  MoveL 9104 to (-26.02, -28.9, -15.5) mm, rotated rx -180 ry 0 rz 90 deg; joints [72.625, -17.388, 85.354, 0, 22.034, 72.625]
  MoveL 9105 to (-25.99, -28.43, -15.5) mm, rotated rx 180 ry 0 rz 90 deg; joints [72.641, -17.39, 85.362, 0, 22.028, 72.641]
  MoveC 9106 to (-26.88, -26.52, -15.5) mm, rotated rx -180 ry 0 rz 90 deg; joints [72.694, -17.416, 85.465, 0, 21.951, 72.694] to (-28.69, -25.44, -15.5) mm, rotated rx 180 ry 0 rz 90 deg; joints [72.71, -17.453, 85.614, 0, 21.839, 72.71]
  MoveL 9107 to (-30.8, -25.8, -15.5) mm, rotated rx 180 ry 0 rz 90 deg; joints [72.677, -17.487, 85.752, 0, 21.735, 72.677]
  MoveL 9108 to (-42.04, -27.96, -15.5) mm, rotated rx 180 ry 0 rz 90 deg; joints [72.492, -17.665, 86.481, 0, 21.184, 72.492]
  MoveL 9109 to (-45.96, -28.7, -15.5) mm, rotated rx -180 ry 0 rz 90 deg; joints [72.427, -17.726, 86.733, 0, 20.993, 72.427]
  MoveL 9110 to (-48.22, -29.15, -15.5) mm, rotated rx -180 ry 0 rz 90 deg; joints [72.389, -17.761, 86.878, 0, 20.882, 72.389]
  MoveL 9111 to (-46.77, -36.56, -15.5) mm, rotated rx -180 ry 0 rz 90 deg; joints [72.161, -17.698, 86.617, 0, 21.081, 72.161]
  MoveL 9112 to (-46.77, -36.56, -12.5) mm, rotated rx -180 ry 0 rz 90 deg; joints [72.161, -17.853, 86.72, 0, 21.133, 72.161]
  Establecer velocidad (1000.0 mm/s)
  MoveL 9113 to (-46.77, -36.56, 10) mm, rotated rx 180 ry 0 rz 90 deg; joints [72.161, -19.016, 87.475, 0, 21.541, 72.161]
  Establecer velocidad (66.7 mm/s)
  MoveL 9114 to (-40.09, -36.12, 10) mm, rotated rx -180 ry 0 rz 90 deg; joints [72.245, -18.904, 87.027, 0, 21.878, 72.245]
  MoveL 9115 to (-40.09, -36.12, -12.5) mm, rotated rx -180 ry 0 rz 90 deg; joints [72.245, -17.744, 86.271, 0, 21.473, 72.245]
  MoveL 9116 to (-40.2, -34.6, -12.91) mm, rotated rx 180 ry 0 rz 90 deg; joints [72.294, -17.733, 86.298, 0, 21.435, 72.294]
  MoveL 9117 to (-40.67, -33.16, -13.31) mm, rotated rx 180 ry 0 rz 90 deg; joints [72.336, -17.728, 86.348, 0, 21.379, 72.336]
  MoveL 9118 to (-41.45, -31.85, -13.72) mm, rotated rx -180 ry 0 rz 90 deg; joints [72.371, -17.727, 86.416, 0, 21.31, 72.371]
  MoveL 9119 to (-42.49, -30.75, -14.12) mm, rotated rx -180 ry 0 rz 90 deg; joints [72.396, -17.729, 86.498, 0, 21.231, 72.396]
  MoveL 9120 to (-43.76, -29.91, -14.53) mm, rotated rx -180 ry 0 rz 90 deg; joints [72.41, -17.733, 86.589, 0, 21.144, 72.41]
  MoveL 9121 to (-45.18, -29.37, -14.94) mm, rotated rx 180 ry 0 rz 90 deg; joints [72.413, -17.739, 86.685, 0, 21.054, 72.413]
  MoveL 9122 to (-46.68, -29.16, -15.34) mm, rotated rx 180 ry 0 rz 90 deg; joints [72.404, -17.743, 86.778, 0, 20.965, 72.404]
  MoveL 9123 to (-48.19, -29.31, -15.75) mm, rotated rx 180 ry 0 rz 90 deg; joints [72.384, -17.746, 86.864, 0, 20.882, 72.384]
  MoveC 9124 to (-48.97, -29.46, -15.75) mm, rotated rx -180 ry 0 rz 90 deg; joints [72.37, -17.758, 86.914, 0, 20.844, 72.37] to (-49.75, -29.62, -15.75) mm, rotated rx 180 ry 0 rz 90 deg; joints [72.357, -17.77, 86.964, 0, 20.807, 72.357]
  MoveL 9125 to (-52.59, -30.15, -15.75) mm, rotated rx -180 ry 0 rz 90 deg; joints [72.31, -17.813, 87.146, 0, 20.668, 72.31]
  MoveL 9126 to (-67.59, -33.11, -15.75) mm, rotated rx 180 ry 0 rz 90 deg; joints [72.054, -18.036, 88.096, 0, 19.939, 72.054]
  MoveC 9127 to (-68.93, -33.88, -15.75) mm, rotated rx -180 ry 0 rz 90 deg; joints [72.014, -18.053, 88.169, 0, 19.883, 72.014] to (-69.53, -35.3, -15.75) mm, rotated rx 180 ry 0 rz 90 deg; joints [71.96, -18.055, 88.179, 0, 19.876, 71.96]
  MoveC 9128 to (-69.55, -35.58, -15.75) mm, rotated rx -180 ry 0 rz 90 deg; joints [71.951, -18.053, 88.174, 0, 19.88, 71.951] to (-69.55, -35.85, -15.75) mm, rotated rx 180 ry 0 rz 90 deg; joints [71.942, -18.052, 88.168, 0, 19.884, 71.942]
  MoveL 9129 to (-69.55, -65.86, -15.75) mm, rotated rx 180 ry 0 rz 90 deg; joints [70.954, -17.895, 87.491, 0, 20.404, 70.954]
  MoveL 9130 to (-69.55, -66.98, -15.75) mm, rotated rx 180 ry 0 rz 90 deg; joints [70.918, -17.889, 87.465, 0, 20.424, 70.918]
  MoveC 9131 to (-68.8, -68.74, -15.75) mm, rotated rx 180 ry 0 rz 90 deg; joints [70.869, -17.867, 87.373, 0, 20.494, 70.869] to (-67.01, -69.45, -15.75) mm, rotated rx 180 ry 0 rz 90 deg; joints [70.866, -17.835, 87.236, 0, 20.599, 70.866]
  MoveC 9132 to (-52.7, -69.11, -15.75) mm, rotated rx -180 ry 0 rz 90 deg; joints [71.037, -17.604, 86.273, 0, 21.33, 71.037] to (-38.38, -68.71, -15.75) mm, rotated rx -180 ry 0 rz 90 deg; joints [71.208, -17.364, 85.301, 0, 22.063, 71.208]
  MoveC 9133 to (-36.78, -68.19, -15.75) mm, rotated rx 180 ry 0 rz 90 deg; joints [71.242, -17.339, 85.203, 0, 22.137, 71.242] to (-35.83, -66.81, -15.75) mm, rotated rx 180 ry 0 rz 90 deg; joints [71.297, -17.331, 85.169, 0, 22.162, 71.297]
  MoveL 9134 to (-26.19, -28.9, -15.75) mm, rotated rx 180 ry 0 rz 90 deg; joints [72.623, -17.378, 85.357, 0, 22.021, 72.623]
  MoveC 9135 to (-26.99, -26.82, -15.75) mm, rotated rx 180 ry 0 rz 90 deg; joints [72.683, -17.403, 85.458, 0, 21.945, 72.683] to (-28.9, -25.65, -15.75) mm, rotated rx 180 ry 0 rz 90 deg; joints [72.701, -17.442, 85.616, 0, 21.827, 72.701]
  MoveC 9136 to (-38.55, -27.45, -15.75) mm, rotated rx -180 ry 0 rz 90 deg; joints [72.544, -17.597, 86.243, 0, 21.353, 72.544] to (-48.19, -29.31, -15.75) mm, rotated rx 180 ry 0 rz 90 deg; joints [72.384, -17.746, 86.864, 0, 20.882, 72.384]
  MoveL 9137 to (-46.74, -36.72, -15.75) mm, rotated rx 180 ry 0 rz 90 deg; joints [72.156, -17.684, 86.603, 0, 21.081, 72.156]
  MoveL 9138 to (-46.74, -36.72, -12.75) mm, rotated rx -180 ry 0 rz 90 deg; joints [72.156, -17.839, 86.705, 0, 21.133, 72.156]
  Establecer velocidad (1000.0 mm/s)
  MoveL 9139 to (-46.74, -36.72, 10) mm, rotated rx 180 ry 0 rz 90 deg; joints [72.156, -19.014, 87.469, 0, 21.545, 72.156]
  Establecer velocidad (66.7 mm/s)
  MoveL 9140 to (-61.31, 35.31, 10) mm, rotated rx -180 ry 0 rz 90 deg; joints [74.405, -19.6, 89.929, 0, 19.671, 74.405]
  MoveL 9141 to (-61.31, 35.31, -12.5) mm, rotated rx -180 ry 0 rz 90 deg; joints [74.405, -18.425, 89.173, 0, 19.251, 74.405]
  MoveL 9142 to (-62.81, 35.49, -12.91) mm, rotated rx 180 ry 0 rz 90 deg; joints [74.397, -18.427, 89.265, 0, 19.162, 74.397]
  MoveL 9143 to (-64.32, 35.31, -13.31) mm, rotated rx 180 ry 0 rz 90 deg; joints [74.377, -18.427, 89.349, 0, 19.079, 74.377]
  MoveL 9144 to (-65.75, 34.8, -13.72) mm, rotated rx -180 ry 0 rz 90 deg; joints [74.346, -18.425, 89.421, 0, 19.004, 74.346]
  MoveL 9145 to (-67.04, 33.98, -14.12) mm, rotated rx -180 ry 0 rz 90 deg; joints [74.306, -18.42, 89.478, 0, 18.941, 74.306]
  MoveL 9146 to (-68.11, 32.9, -14.53) mm, rotated rx 180 ry 0 rz 90 deg; joints [74.259, -18.41, 89.516, 0, 18.894, 74.259]
  MoveL 9147 to (-68.91, 31.61, -14.94) mm, rotated rx -180 ry 0 rz 90 deg; joints [74.208, -18.395, 89.531, 0, 18.864, 74.208]
  MoveL 9148 to (-69.41, 30.18, -15.34) mm, rotated rx 180 ry 0 rz 90 deg; joints [74.154, -18.375, 89.524, 0, 18.851, 74.154]
  MoveL 9149 to (-69.55, 28.67, -15.75) mm, rotated rx 180 ry 0 rz 90 deg; joints [74.102, -18.349, 89.49, 0, 18.859, 74.102]
  MoveL 9150 to (-69.55, 5.69, -15.75) mm, rotated rx -180 ry 0 rz 90 deg; joints [73.327, -18.25, 89.04, 0, 19.21, 73.327]
  MoveC 9151 to (-68.75, 3.78, -15.75) mm, rotated rx 180 ry 0 rz 90 deg; joints [73.271, -18.229, 88.948, 0, 19.281, 73.271] to (-66.81, 3.09, -15.75) mm, rotated rx 180 ry 0 rz 90 deg; joints [73.267, -18.197, 88.804, 0, 19.393, 73.267]
  MoveL 9152 to (-65.86, 3.29, -15.75) mm, rotated rx 180 ry 0 rz 90 deg; joints [73.283, -18.183, 88.744, 0, 19.439, 73.283]
  MoveL 9153 to (-62.19, 4.19, -15.75) mm, rotated rx -180 ry 0 rz 90 deg; joints [73.35, -18.131, 88.515, 0, 19.616, 73.35]
  MoveC 9154 to (-44.56, 8.55, -15.75) mm, rotated rx 180 ry 0 rz 90 deg; joints [73.67, -17.875, 87.406, 0, 20.469, 73.67] to (-26.96, 13.02, -15.75) mm, rotated rx 180 ry 0 rz 90 deg; joints [73.986, -17.606, 86.283, 0, 21.323, 73.986]
  MoveC 9155 to (-26.48, 13.21, -15.75) mm, rotated rx -180 ry 0 rz 90 deg; joints [73.997, -17.599, 86.254, 0, 21.345, 73.997] to (-26.06, 13.5, -15.75) mm, rotated rx 180 ry 0 rz 90 deg; joints [74.01, -17.593, 86.231, 0, 21.363, 74.01]
  MoveC 9156 to (-25.23, 14.68, -15.75) mm, rotated rx -180 ry 0 rz 90 deg; joints [74.057, -17.585, 86.197, 0, 21.389, 74.057] to (-25.03, 16.11, -15.75) mm, rotated rx 180 ry 0 rz 90 deg; joints [74.106, -17.589, 86.211, 0, 21.378, 74.106]
  MoveC 9157 to (-25.09, 16.38, -15.75) mm, rotated rx 180 ry 0 rz 90 deg; joints [74.114, -17.591, 86.22, 0, 21.371, 74.114] to (-25.17, 16.64, -15.75) mm, rotated rx 180 ry 0 rz 90 deg; joints [74.122, -17.594, 86.231, 0, 21.362, 74.122]
  MoveL 9158 to (-29.47, 28.93, -15.75) mm, rotated rx -180 ry 0 rz 90 deg; joints [74.488, -17.723, 86.768, 0, 20.955, 74.488]
  MoveC 9159 to (-29.9, 29.71, -15.75) mm, rotated rx 180 ry 0 rz 90 deg; joints [74.51, -17.734, 86.812, 0, 20.922, 74.51] to (-30.55, 30.32, -15.75) mm, rotated rx 180 ry 0 rz 90 deg; joints [74.525, -17.747, 86.869, 0, 20.879, 74.525]
  MoveC 9160 to (-48.17, 42.1, -15.75) mm, rotated rx 180 ry 0 rz 90 deg; joints [74.756, -18.082, 88.299, 0, 19.783, 74.756] to (-65.86, 53.77, -15.75) mm, rotated rx 180 ry 0 rz 90 deg; joints [74.989, -18.397, 89.708, 0, 18.689, 74.989]
  MoveC 9161 to (-67.73, 53.7, -15.75) mm, rotated rx 180 ry 0 rz 90 deg; joints [74.97, -18.424, 89.832, 0, 18.592, 74.97] to (-69.23, 52.59, -15.75) mm, rotated rx 180 ry 0 rz 90 deg; joints [74.918, -18.442, 89.913, 0, 18.529, 74.918]
  MoveC 9162 to (-69.47, 52.15, -15.75) mm, rotated rx 180 ry 0 rz 90 deg; joints [74.901, -18.443, 89.921, 0, 18.522, 74.901] to (-69.55, 51.65, -15.75) mm, rotated rx 180 ry 0 rz 90 deg; joints [74.883, -18.442, 89.917, 0, 18.525, 74.883]
  MoveL 9163 to (-69.55, 28.67, -15.75) mm, rotated rx 180 ry 0 rz 90 deg; joints [74.102, -18.349, 89.49, 0, 18.859, 74.102]
  MoveL 9164 to (-62, 28.67, -15.75) mm, rotated rx -180 ry 0 rz 90 deg; joints [74.174, -18.237, 88.983, 0, 19.254, 74.174]
  MoveL 9165 to (-62, 28.67, -12.75) mm, rotated rx 180 ry 0 rz 90 deg; joints [74.174, -18.394, 89.086, 0, 19.308, 74.174]
  Establecer velocidad (1000.0 mm/s)
  MoveL 9166 to (-62, 28.67, 10) mm, rotated rx 180 ry 0 rz 90 deg; joints [74.174, -19.582, 89.85, 0, 19.732, 74.174]
  Establecer velocidad (66.7 mm/s)
  MoveL 9167 to (-61.15, 35.31, 10) mm, rotated rx 180 ry 0 rz 90 deg; joints [74.407, -19.598, 89.918, 0, 19.679, 74.407]
  MoveL 9168 to (-61.15, 35.31, -12.75) mm, rotated rx 180 ry 0 rz 90 deg; joints [74.407, -18.409, 89.154, 0, 19.255, 74.407]
  MoveL 9169 to (-62.65, 35.49, -13.16) mm, rotated rx -180 ry 0 rz 90 deg; joints [74.399, -18.411, 89.245, 0, 19.166, 74.399]
  MoveL 9170 to (-64.16, 35.31, -13.56) mm, rotated rx 180 ry 0 rz 90 deg; joints [74.378, -18.412, 89.329, 0, 19.083, 74.378]
  MoveL 9171 to (-65.59, 34.8, -13.97) mm, rotated rx -180 ry 0 rz 90 deg; joints [74.347, -18.41, 89.402, 0, 19.008, 74.347]
  MoveL 9172 to (-66.87, 33.98, -14.37) mm, rotated rx 180 ry 0 rz 90 deg; joints [74.308, -18.404, 89.459, 0, 18.945, 74.308]
  MoveL 9173 to (-67.94, 32.9, -14.78) mm, rotated rx -180 ry 0 rz 90 deg; joints [74.261, -18.394, 89.496, 0, 18.898, 74.261]
  MoveL 9174 to (-68.75, 31.61, -15.19) mm, rotated rx -180 ry 0 rz 90 deg; joints [74.209, -18.379, 89.512, 0, 18.868, 74.209]
  MoveL 9175 to (-69.25, 30.18, -15.59) mm, rotated rx 180 ry 0 rz 90 deg; joints [74.156, -18.359, 89.504, 0, 18.856, 74.156]
  MoveL 9176 to (-69.39, 28.67, -16) mm, rotated rx -180 ry 0 rz 90 deg; joints [74.104, -18.334, 89.471, 0, 18.863, 74.104]
  MoveL 9177 to (-69.39, 6.16, -16) mm, rotated rx -180 ry 0 rz 90 deg; joints [73.344, -18.236, 89.03, 0, 19.206, 73.344]
  MoveL 9178 to (-69.38, 5.69, -16) mm, rotated rx -180 ry 0 rz 90 deg; joints [73.329, -18.234, 89.02, 0, 19.214, 73.329]
  MoveC 9179 to (-68.41, 3.79, -16) mm, rotated rx -180 ry 0 rz 90 deg; joints [73.275, -18.211, 88.917, 0, 19.294, 73.275] to (-66.33, 3.32, -16) mm, rotated rx 180 ry 0 rz 90 deg; joints [73.28, -18.178, 88.768, 0, 19.41, 73.28]
  MoveC 9180 to (-46.77, 8.15, -16) mm, rotated rx 180 ry 0 rz 90 deg; joints [73.635, -17.895, 87.54, 0, 20.356, 73.635] to (-27.23, 13.12, -16) mm, rotated rx 180 ry 0 rz 90 deg; joints [73.987, -17.598, 86.296, 0, 21.303, 73.987]
  MoveC 9181 to (-26.84, 13.26, -16) mm, rotated rx 180 ry 0 rz 90 deg; joints [73.995, -17.592, 86.271, 0, 21.322, 73.995] to (-26.47, 13.45, -16) mm, rotated rx -180 ry 0 rz 90 deg; joints [74.005, -17.587, 86.249, 0, 21.338, 74.005]
  MoveC 9182 to (-25.52, 14.63, -16) mm, rotated rx -180 ry 0 rz 90 deg; joints [74.053, -17.577, 86.206, 0, 21.37, 74.053] to (-25.22, 16.11, -16) mm, rotated rx 180 ry 0 rz 90 deg; joints [74.104, -17.579, 86.215, 0, 21.364, 74.104]
  MoveC 9183 to (-25.32, 16.55, -16) mm, rotated rx 180 ry 0 rz 90 deg; joints [74.118, -17.583, 86.231, 0, 21.352, 74.118] to (-25.46, 16.98, -16) mm, rotated rx -180 ry 0 rz 90 deg; joints [74.131, -17.587, 86.249, 0, 21.338, 74.131]
  MoveL 9184 to (-25.99, 18.48, -16) mm, rotated rx 180 ry 0 rz 90 deg; joints [74.175, -17.603, 86.315, 0, 21.288, 74.175]
  MoveL 9185 to (-29.61, 28.86, -16) mm, rotated rx -180 ry 0 rz 90 deg; joints [74.485, -17.712, 86.767, 0, 20.945, 74.485]
  MoveC 9186 to (-30.01, 29.61, -16) mm, rotated rx -180 ry 0 rz 90 deg; joints [74.506, -17.723, 86.81, 0, 20.913, 74.506] to (-30.64, 30.19, -16) mm, rotated rx 180 ry 0 rz 90 deg; joints [74.519, -17.736, 86.864, 0, 20.872, 74.519]
  MoveC 9187 to (-48.16, 41.92, -16) mm, rotated rx 180 ry 0 rz 90 deg; joints [74.75, -18.068, 88.287, 0, 19.782, 74.75] to (-65.76, 53.54, -16) mm, rotated rx 180 ry 0 rz 90 deg; joints [74.983, -18.382, 89.689, 0, 18.693, 74.983]
  MoveC 9188 to (-67.74, 53.4, -16) mm, rotated rx -180 ry 0 rz 90 deg; joints [74.96, -18.41, 89.819, 0, 18.591, 74.96] to (-69.23, 52.1, -16) mm, rotated rx 180 ry 0 rz 90 deg; joints [74.901, -18.427, 89.895, 0, 18.531, 74.901]
  MoveC 9189 to (-69.34, 51.82, -16) mm, rotated rx 180 ry 0 rz 90 deg; joints [74.891, -18.427, 89.898, 0, 18.529, 74.891] to (-69.39, 51.53, -16) mm, rotated rx 180 ry 0 rz 90 deg; joints [74.881, -18.427, 89.896, 0, 18.531, 74.881]
  MoveL 9190 to (-69.39, 28.67, -16) mm, rotated rx -180 ry 0 rz 90 deg; joints [74.104, -18.334, 89.471, 0, 18.863, 74.104]
  MoveL 9191 to (-61.84, 28.67, -16) mm, rotated rx 180 ry 0 rz 90 deg; joints [74.176, -18.221, 88.963, 0, 19.258, 74.176]
  MoveL 9192 to (-61.84, 28.67, -13) mm, rotated rx -180 ry 0 rz 90 deg; joints [74.176, -18.378, 89.066, 0, 19.312, 74.176]
  Establecer velocidad (1000.0 mm/s)
  MoveL 9193 to (-61.84, 28.67, 10) mm, rotated rx 180 ry 0 rz 90 deg; joints [74.176, -19.58, 89.839, 0, 19.741, 74.176]
  Establecer velocidad (66.7 mm/s)
  MoveL 9194 to (-40.16, -36.29, 10) mm, rotated rx 180 ry 0 rz 90 deg; joints [72.239, -18.905, 87.028, 0, 21.877, 72.239]
  MoveL 9195 to (-40.16, -36.29, -12.75) mm, rotated rx 180 ry 0 rz 90 deg; joints [72.239, -17.731, 86.264, 0, 21.467, 72.239]
  MoveL 9196 to (-40.27, -34.78, -13.16) mm, rotated rx 180 ry 0 rz 90 deg; joints [72.287, -17.72, 86.291, 0, 21.429, 72.287]
  MoveL 9197 to (-40.74, -33.33, -13.56) mm, rotated rx 180 ry 0 rz 90 deg; joints [72.33, -17.715, 86.341, 0, 21.374, 72.33]
  MoveL 9198 to (-41.52, -32.02, -13.97) mm, rotated rx 180 ry 0 rz 90 deg; joints [72.364, -17.714, 86.409, 0, 21.305, 72.364]
  MoveL 9199 to (-42.57, -30.92, -14.37) mm, rotated rx 180 ry 0 rz 90 deg; joints [72.389, -17.717, 86.491, 0, 21.225, 72.389]
  MoveL 9200 to (-43.84, -30.09, -14.78) mm, rotated rx 180 ry 0 rz 90 deg; joints [72.403, -17.721, 86.583, 0, 21.138, 72.403]
  MoveL 9201 to (-45.26, -29.55, -15.19) mm, rotated rx 180 ry 0 rz 90 deg; joints [72.406, -17.726, 86.678, 0, 21.049, 72.406]
  MoveL 9202 to (-46.77, -29.33, -15.59) mm, rotated rx -180 ry 0 rz 90 deg; joints [72.398, -17.731, 86.771, 0, 20.96, 72.398]
  MoveL 9203 to (-48.28, -29.49, -16) mm, rotated rx 180 ry 0 rz 90 deg; joints [72.377, -17.734, 86.857, 0, 20.877, 72.377]
  MoveL 9204 to (-49.75, -29.78, -16) mm, rotated rx 180 ry 0 rz 90 deg; joints [72.352, -17.756, 86.952, 0, 20.805, 72.352]
  MoveL 9205 to (-52.59, -30.31, -16) mm, rotated rx -180 ry 0 rz 90 deg; joints [72.305, -17.8, 87.134, 0, 20.666, 72.305]
  MoveL 9206 to (-67.44, -33.23, -16) mm, rotated rx 180 ry 0 rz 90 deg; joints [72.051, -18.02, 88.075, 0, 19.945, 72.051]
  MoveC 9207 to (-68.76, -33.98, -16) mm, rotated rx -180 ry 0 rz 90 deg; joints [72.012, -18.036, 88.147, 0, 19.889, 72.012] to (-69.36, -35.37, -16) mm, rotated rx -180 ry 0 rz 90 deg; joints [71.96, -18.039, 88.157, 0, 19.881, 71.96]
  MoveC 9208 to (-69.38, -35.65, -16) mm, rotated rx 180 ry 0 rz 90 deg; joints [71.95, -18.038, 88.152, 0, 19.885, 71.95] to (-69.39, -35.94, -16) mm, rotated rx -180 ry 0 rz 90 deg; joints [71.94, -18.036, 88.146, 0, 19.89, 71.94]
  MoveL 9209 to (-69.39, -65.86, -16) mm, rotated rx 180 ry 0 rz 90 deg; joints [70.956, -17.879, 87.471, 0, 20.408, 70.956]
  MoveL 9210 to (-69.38, -66.81, -16) mm, rotated rx -180 ry 0 rz 90 deg; joints [70.925, -17.874, 87.449, 0, 20.425, 70.925]
  MoveC 9211 to (-68.63, -68.61, -16) mm, rotated rx 180 ry 0 rz 90 deg; joints [70.875, -17.852, 87.356, 0, 20.496, 70.875] to (-66.81, -69.3, -16) mm, rotated rx 180 ry 0 rz 90 deg; joints [70.873, -17.82, 87.218, 0, 20.602, 70.873]
  MoveC 9212 to (-52.58, -68.96, -16) mm, rotated rx -180 ry 0 rz 90 deg; joints [71.044, -17.59, 86.26, 0, 21.33, 71.044] to (-38.35, -68.54, -16) mm, rotated rx 180 ry 0 rz 90 deg; joints [71.214, -17.352, 85.294, 0, 22.058, 71.214]
  MoveC 9213 to (-36.8, -67.97, -16) mm, rotated rx 180 ry 0 rz 90 deg; joints [71.249, -17.328, 85.201, 0, 22.128, 71.249] to (-35.92, -66.59, -16) mm, rotated rx -180 ry 0 rz 90 deg; joints [71.304, -17.321, 85.172, 0, 22.149, 71.304]
  MoveL 9214 to (-26.47, -29.38, -16) mm, rotated rx -180 ry 0 rz 90 deg; joints [72.605, -17.367, 85.357, 0, 22.01, 72.605]
  MoveC 9215 to (-26.5, -28.28, -16) mm, rotated rx -180 ry 0 rz 90 deg; joints [72.64, -17.374, 85.383, 0, 21.991, 72.64] to (-27.01, -27.31, -16) mm, rotated rx -180 ry 0 rz 90 deg; joints [72.667, -17.388, 85.44, 0, 21.948, 72.667]
  MoveC 9216 to (-27.9, -26.37, -16) mm, rotated rx -180 ry 0 rz 90 deg; joints [72.688, -17.408, 85.522, 0, 21.887, 72.688] to (-29.09, -25.87, -16) mm, rotated rx 180 ry 0 rz 90 deg; joints [72.692, -17.432, 85.615, 0, 21.816, 72.692]
  MoveL 9217 to (-30.33, -26.08, -16) mm, rotated rx 180 ry 0 rz 90 deg; joints [72.673, -17.452, 85.696, 0, 21.755, 72.673]
  MoveL 9218 to (-45.96, -29.03, -16) mm, rotated rx 180 ry 0 rz 90 deg; joints [72.416, -17.698, 86.709, 0, 20.989, 72.416]
  MoveL 9219 to (-48.28, -29.49, -16) mm, rotated rx 180 ry 0 rz 90 deg; joints [72.377, -17.734, 86.857, 0, 20.877, 72.377]
  MoveL 9220 to (-46.81, -36.9, -16) mm, rotated rx 180 ry 0 rz 90 deg; joints [72.15, -17.671, 86.595, 0, 21.076, 72.15]
  MoveL 9221 to (-46.81, -36.9, -13) mm, rotated rx 180 ry 0 rz 90 deg; joints [72.15, -17.826, 86.698, 0, 21.128, 72.15]
  Establecer velocidad (1000.0 mm/s)
  MoveL 9222 to (-46.81, -36.9, 10) mm, rotated rx -180 ry 0 rz 90 deg; joints [72.15, -19.015, 87.47, 0, 21.544, 72.15]
  Establecer velocidad (66.7 mm/s)
  MoveL 9223 to (-40.18, -36.49, 10) mm, rotated rx 180 ry 0 rz 90 deg; joints [72.233, -18.904, 87.025, 0, 21.879, 72.233]
  MoveL 9224 to (-40.18, -36.49, -13) mm, rotated rx -180 ry 0 rz 90 deg; joints [72.233, -17.718, 86.252, 0, 21.466, 72.233]
  MoveL 9225 to (-40.28, -34.97, -13.41) mm, rotated rx 180 ry 0 rz 90 deg; joints [72.281, -17.707, 86.278, 0, 21.428, 72.281]
  MoveL 9226 to (-40.74, -33.53, -13.81) mm, rotated rx -180 ry 0 rz 90 deg; joints [72.323, -17.701, 86.328, 0, 21.373, 72.323]
  MoveL 9227 to (-41.51, -32.22, -14.22) mm, rotated rx -180 ry 0 rz 90 deg; joints [72.358, -17.7, 86.396, 0, 21.304, 72.358]
  MoveL 9228 to (-42.56, -31.11, -14.63) mm, rotated rx 180 ry 0 rz 90 deg; joints [72.383, -17.702, 86.478, 0, 21.225, 72.383]
  MoveL 9229 to (-43.82, -30.26, -15.03) mm, rotated rx -180 ry 0 rz 90 deg; joints [72.398, -17.707, 86.568, 0, 21.138, 72.398]
  MoveL 9230 to (-45.23, -29.72, -15.44) mm, rotated rx -180 ry 0 rz 90 deg; joints [72.401, -17.712, 86.663, 0, 21.048, 72.401]
  MoveL 9231 to (-46.74, -29.49, -15.84) mm, rotated rx -180 ry 0 rz 90 deg; joints [72.393, -17.717, 86.757, 0, 20.959, 72.393]
  MoveL 9232 to (-48.25, -29.64, -16.25) mm, rotated rx -180 ry 0 rz 90 deg; joints [72.372, -17.72, 86.843, 0, 20.876, 72.372]
  MoveC 9233 to (-57.78, -31.48, -16.25) mm, rotated rx 180 ry 0 rz 90 deg; joints [72.212, -17.864, 87.452, 0, 20.412, 72.212] to (-67.32, -33.36, -16.25) mm, rotated rx -180 ry 0 rz 90 deg; joints [72.048, -18.004, 88.055, 0, 19.949, 72.048]
  MoveC 9234 to (-68.58, -34.07, -16.25) mm, rotated rx 180 ry 0 rz 90 deg; joints [72.011, -18.02, 88.125, 0, 19.895, 72.011] to (-69.19, -35.39, -16.25) mm, rotated rx 180 ry 0 rz 90 deg; joints [71.961, -18.023, 88.137, 0, 19.886, 71.961]
  MoveC 9235 to (-69.21, -35.68, -16.25) mm, rotated rx 180 ry 0 rz 90 deg; joints [71.951, -18.022, 88.132, 0, 19.89, 71.951] to (-69.22, -35.97, -16.25) mm, rotated rx -180 ry 0 rz 90 deg; joints [71.941, -18.02, 88.126, 0, 19.894, 71.941]
  MoveL 9236 to (-69.22, -65.86, -16.25) mm, rotated rx 180 ry 0 rz 90 deg; joints [70.958, -17.864, 87.452, 0, 20.412, 70.958]
  MoveL 9237 to (-69.21, -66.81, -16.25) mm, rotated rx 180 ry 0 rz 90 deg; joints [70.927, -17.858, 87.429, 0, 20.43, 70.927]
  MoveC 9238 to (-68.48, -68.47, -16.25) mm, rotated rx -180 ry 0 rz 90 deg; joints [70.881, -17.838, 87.341, 0, 20.497, 70.881] to (-66.81, -69.15, -16.25) mm, rotated rx 180 ry 0 rz 90 deg; joints [70.878, -17.807, 87.212, 0, 20.595, 70.878]
  MoveC 9239 to (-52.59, -68.81, -16.25) mm, rotated rx -180 ry 0 rz 90 deg; joints [71.048, -17.578, 86.256, 0, 21.322, 71.048] to (-38.38, -68.37, -16.25) mm, rotated rx 180 ry 0 rz 90 deg; joints [71.219, -17.34, 85.291, 0, 22.049, 71.219]
  MoveC 9240 to (-36.85, -67.77, -16.25) mm, rotated rx 180 ry 0 rz 90 deg; joints [71.255, -17.317, 85.2, 0, 22.117, 71.255] to (-36.01, -66.36, -16.25) mm, rotated rx 180 ry 0 rz 90 deg; joints [71.31, -17.311, 85.175, 0, 22.136, 71.31]
  MoveL 9241 to (-26.7, -29.65, -16.25) mm, rotated rx -180 ry 0 rz 90 deg; joints [72.594, -17.357, 85.359, 0, 21.998, 72.594]
  MoveC 9242 to (-26.64, -29.28, -16.25) mm, rotated rx 180 ry 0 rz 90 deg; joints [72.606, -17.358, 85.362, 0, 21.996, 72.606] to (-26.63, -28.9, -16.25) mm, rotated rx 180 ry 0 rz 90 deg; joints [72.619, -17.36, 85.37, 0, 21.99, 72.619]
  MoveC 9243 to (-27.5, -27.13, -16.25) mm, rotated rx 180 ry 0 rz 90 deg; joints [72.667, -17.384, 85.469, 0, 21.915, 72.667] to (-29.17, -26.09, -16.25) mm, rotated rx -180 ry 0 rz 90 deg; joints [72.684, -17.419, 85.608, 0, 21.811, 72.684]
  MoveL 9244 to (-29.38, -26.1, -16.25) mm, rotated rx 180 ry 0 rz 90 deg; joints [72.682, -17.422, 85.622, 0, 21.801, 72.682]
  MoveL 9245 to (-30.03, -26.22, -16.25) mm, rotated rx -180 ry 0 rz 90 deg; joints [72.671, -17.433, 85.664, 0, 21.769, 72.671]
  MoveC 9246 to (-39.14, -27.92, -16.25) mm, rotated rx -180 ry 0 rz 90 deg; joints [72.523, -17.578, 86.256, 0, 21.322, 72.523] to (-48.25, -29.64, -16.25) mm, rotated rx -180 ry 0 rz 90 deg; joints [72.372, -17.72, 86.843, 0, 20.876, 72.372]
  MoveL 9247 to (-46.83, -37.06, -16.25) mm, rotated rx 180 ry 0 rz 90 deg; joints [72.144, -17.657, 86.584, 0, 21.073, 72.144]
  MoveL 9248 to (-46.83, -37.06, -13.25) mm, rotated rx -180 ry 0 rz 90 deg; joints [72.144, -17.813, 86.687, 0, 21.126, 72.144]
  Establecer velocidad (1000.0 mm/s)
  MoveL 9249 to (-46.83, -37.06, 10) mm, rotated rx -180 ry 0 rz 90 deg; joints [72.144, -19.014, 87.468, 0, 21.546, 72.144]
  Establecer velocidad (66.7 mm/s)
  MoveL 9250 to (-60.98, 35.19, 10) mm, rotated rx -180 ry 0 rz 90 deg; joints [74.404, -19.595, 89.905, 0, 19.69, 74.404]
  MoveL 9251 to (-60.98, 35.19, -13) mm, rotated rx 180 ry 0 rz 90 deg; joints [74.404, -18.393, 89.132, 0, 19.261, 74.404]
  MoveL 9252 to (-62.49, 35.37, -13.41) mm, rotated rx 180 ry 0 rz 90 deg; joints [74.396, -18.395, 89.223, 0, 19.172, 74.396]
  MoveL 9253 to (-64, 35.19, -13.81) mm, rotated rx 180 ry 0 rz 90 deg; joints [74.376, -18.396, 89.307, 0, 19.088, 74.376]
  MoveL 9254 to (-65.43, 34.68, -14.22) mm, rotated rx -180 ry 0 rz 90 deg; joints [74.345, -18.394, 89.38, 0, 19.014, 74.345]
  MoveL 9255 to (-66.71, 33.86, -14.63) mm, rotated rx -180 ry 0 rz 90 deg; joints [74.305, -18.388, 89.437, 0, 18.951, 74.305]
  MoveL 9256 to (-67.78, 32.78, -15.03) mm, rotated rx -180 ry 0 rz 90 deg; joints [74.258, -18.378, 89.474, 0, 18.904, 74.258]
  MoveL 9257 to (-68.58, 31.49, -15.44) mm, rotated rx 180 ry 0 rz 90 deg; joints [74.207, -18.363, 89.49, 0, 18.874, 74.207]
  MoveL 9258 to (-69.08, 30.06, -15.84) mm, rotated rx 180 ry 0 rz 90 deg; joints [74.154, -18.343, 89.482, 0, 18.861, 74.154]
  MoveL 9259 to (-69.22, 28.55, -16.25) mm, rotated rx 180 ry 0 rz 90 deg; joints [74.101, -18.318, 89.449, 0, 18.869, 74.101]
  MoveL 9260 to (-69.22, 5.91, -16.25) mm, rotated rx 180 ry 0 rz 90 deg; joints [73.338, -18.22, 89.005, 0, 19.214, 73.338]
  MoveC 9261 to (-68.29, 3.98, -16.25) mm, rotated rx -180 ry 0 rz 90 deg; joints [73.282, -18.197, 88.904, 0, 19.293, 73.282] to (-66.21, 3.5, -16.25) mm, rotated rx -180 ry 0 rz 90 deg; joints [73.287, -18.163, 88.754, 0, 19.409, 73.287]
  MoveL 9262 to (-65.86, 3.58, -16.25) mm, rotated rx 180 ry 0 rz 90 deg; joints [73.293, -18.158, 88.733, 0, 19.426, 73.293]
  MoveC 9263 to (-46.6, 8.35, -16.25) mm, rotated rx 180 ry 0 rz 90 deg; joints [73.643, -17.881, 87.524, 0, 20.357, 73.643] to (-27.38, 13.27, -16.25) mm, rotated rx 180 ry 0 rz 90 deg; joints [73.99, -17.589, 86.3, 0, 21.289, 73.99]
  MoveC 9264 to (-26.63, 13.6, -16.25) mm, rotated rx -180 ry 0 rz 90 deg; joints [74.008, -17.578, 86.255, 0, 21.323, 74.008] to (-26.06, 14.19, -16.25) mm, rotated rx -180 ry 0 rz 90 deg; joints [74.033, -17.571, 86.227, 0, 21.344, 74.033]
  MoveC 9265 to (-25.51, 15.32, -16.25) mm, rotated rx 180 ry 0 rz 90 deg; joints [74.076, -17.567, 86.211, 0, 21.356, 74.076] to (-25.51, 16.58, -16.25) mm, rotated rx -180 ry 0 rz 90 deg; joints [74.117, -17.573, 86.236, 0, 21.337, 74.117]
  MoveL 9266 to (-29.74, 28.76, -16.25) mm, rotated rx 180 ry 0 rz 90 deg; joints [74.48, -17.701, 86.766, 0, 20.935, 74.48]
  MoveC 9267 to (-30.14, 29.49, -16.25) mm, rotated rx 180 ry 0 rz 90 deg; joints [74.501, -17.711, 86.807, 0, 20.904, 74.501] to (-30.74, 30.07, -16.25) mm, rotated rx -180 ry 0 rz 90 deg; joints [74.514, -17.724, 86.86, 0, 20.863, 74.514]
  MoveC 9268 to (-48.17, 41.75, -16.25) mm, rotated rx -180 ry 0 rz 90 deg; joints [74.744, -18.055, 88.275, 0, 19.779, 74.744] to (-65.67, 53.31, -16.25) mm, rotated rx -180 ry 0 rz 90 deg; joints [74.976, -18.366, 89.67, 0, 18.696, 74.976]
  MoveC 9269 to (-67.48, 53.2, -16.25) mm, rotated rx -180 ry 0 rz 90 deg; joints [74.955, -18.392, 89.79, 0, 18.603, 74.955] to (-68.93, 52.09, -16.25) mm, rotated rx 180 ry 0 rz 90 deg; joints [74.904, -18.409, 89.866, 0, 18.543, 74.904]
  MoveC 9270 to (-69.15, 51.66, -16.25) mm, rotated rx 180 ry 0 rz 90 deg; joints [74.887, -18.41, 89.873, 0, 18.537, 74.887] to (-69.22, 51.18, -16.25) mm, rotated rx -180 ry 0 rz 90 deg; joints [74.87, -18.41, 89.87, 0, 18.54, 74.87]
  MoveL 9271 to (-69.22, 28.55, -16.25) mm, rotated rx 180 ry 0 rz 90 deg; joints [74.101, -18.318, 89.449, 0, 18.869, 74.101]
  MoveL 9272 to (-61.67, 28.55, -16.25) mm, rotated rx 180 ry 0 rz 90 deg; joints [74.174, -18.205, 88.941, 0, 19.264, 74.174]
  MoveL 9273 to (-61.67, 28.55, -13.25) mm, rotated rx -180 ry 0 rz 90 deg; joints [74.174, -18.362, 89.044, 0, 19.318, 74.174]
  Establecer velocidad (1000.0 mm/s)
  MoveL 9274 to (-61.67, 28.55, 10) mm, rotated rx -180 ry 0 rz 90 deg; joints [74.174, -19.576, 89.826, 0, 19.751, 74.174]
  Establecer velocidad (66.7 mm/s)
  MoveL 9275 to (-60.82, 35.19, 10) mm, rotated rx -180 ry 0 rz 90 deg; joints [74.406, -19.592, 89.894, 0, 19.698, 74.406]
  MoveL 9276 to (-60.82, 35.19, -13.25) mm, rotated rx 180 ry 0 rz 90 deg; joints [74.406, -18.377, 89.112, 0, 19.265, 74.406]
  MoveL 9277 to (-62.32, 35.37, -13.66) mm, rotated rx 180 ry 0 rz 90 deg; joints [74.398, -18.38, 89.203, 0, 19.176, 74.398]
  MoveL 9278 to (-63.83, 35.19, -14.06) mm, rotated rx -180 ry 0 rz 90 deg; joints [74.377, -18.38, 89.288, 0, 19.093, 74.377]
  MoveL 9279 to (-65.26, 34.68, -14.47) mm, rotated rx 180 ry 0 rz 90 deg; joints [74.346, -18.378, 89.36, 0, 19.018, 74.346]
  MoveL 9280 to (-66.54, 33.86, -14.87) mm, rotated rx 180 ry 0 rz 90 deg; joints [74.307, -18.373, 89.417, 0, 18.955, 74.307]
  MoveL 9281 to (-67.61, 32.78, -15.28) mm, rotated rx 180 ry 0 rz 90 deg; joints [74.26, -18.363, 89.455, 0, 18.908, 74.26]
  MoveL 9282 to (-68.42, 31.49, -15.69) mm, rotated rx -180 ry 0 rz 90 deg; joints [74.209, -18.348, 89.47, 0, 18.878, 74.209]
  MoveL 9283 to (-68.92, 30.06, -16.09) mm, rotated rx 180 ry 0 rz 90 deg; joints [74.155, -18.328, 89.462, 0, 18.865, 74.155]
  MoveL 9284 to (-69.06, 28.55, -16.5) mm, rotated rx -180 ry 0 rz 90 deg; joints [74.103, -18.302, 89.429, 0, 18.873, 74.103]
  MoveL 9285 to (-69.05, 6.16, -16.5) mm, rotated rx 180 ry 0 rz 90 deg; joints [73.348, -18.205, 88.991, 0, 19.215, 73.348]
  MoveC 9286 to (-68.27, 4.27, -16.5) mm, rotated rx -180 ry 0 rz 90 deg; joints [73.292, -18.185, 88.9, 0, 19.285, 73.292] to (-66.33, 3.62, -16.5) mm, rotated rx -180 ry 0 rz 90 deg; joints [73.29, -18.153, 88.757, 0, 19.396, 73.29]
  MoveL 9287 to (-65.86, 3.72, -16.5) mm, rotated rx 180 ry 0 rz 90 deg; joints [73.298, -18.146, 88.727, 0, 19.419, 73.298]
  MoveC 9288 to (-46.71, 8.48, -16.5) mm, rotated rx 180 ry 0 rz 90 deg; joints [73.646, -17.87, 87.525, 0, 20.345, 73.646] to (-27.6, 13.38, -16.5) mm, rotated rx 180 ry 0 rz 90 deg; joints [73.992, -17.58, 86.309, 0, 21.271, 73.992]
  MoveC 9289 to (-26.7, 13.83, -16.5) mm, rotated rx -180 ry 0 rz 90 deg; joints [74.015, -17.567, 86.256, 0, 21.311, 74.015] to (-26.06, 14.59, -16.5) mm, rotated rx -180 ry 0 rz 90 deg; joints [74.046, -17.56, 86.226, 0, 21.334, 74.046]
  MoveC 9290 to (-25.66, 15.67, -16.5) mm, rotated rx 180 ry 0 rz 90 deg; joints [74.086, -17.558, 86.22, 0, 21.339, 74.086] to (-25.76, 16.81, -16.5) mm, rotated rx 180 ry 0 rz 90 deg; joints [74.122, -17.565, 86.249, 0, 21.316, 74.122]
  MoveL 9291 to (-25.98, 17.53, -16.5) mm, rotated rx -180 ry 0 rz 90 deg; joints [74.144, -17.573, 86.279, 0, 21.294, 74.144]
  MoveL 9292 to (-29.85, 28.62, -16.5) mm, rotated rx 180 ry 0 rz 90 deg; joints [74.475, -17.689, 86.762, 0, 20.927, 74.475]
  MoveC 9293 to (-30.22, 29.34, -16.5) mm, rotated rx -180 ry 0 rz 90 deg; joints [74.495, -17.699, 86.802, 0, 20.897, 74.495] to (-30.8, 29.91, -16.5) mm, rotated rx -180 ry 0 rz 90 deg; joints [74.508, -17.711, 86.852, 0, 20.859, 74.508]
  MoveC 9294 to (-48.13, 41.55, -16.5) mm, rotated rx -180 ry 0 rz 90 deg; joints [74.738, -18.04, 88.26, 0, 19.78, 74.738] to (-65.54, 53.07, -16.5) mm, rotated rx -180 ry 0 rz 90 deg; joints [74.968, -18.35, 89.648, 0, 18.702, 74.968]
  MoveC 9295 to (-67.3, 52.96, -16.5) mm, rotated rx 180 ry 0 rz 90 deg; joints [74.949, -18.376, 89.764, 0, 18.611, 74.949] to (-68.73, 51.93, -16.5) mm, rotated rx 180 ry 0 rz 90 deg; joints [74.9, -18.392, 89.841, 0, 18.551, 74.9]
  MoveC 9296 to (-68.97, 51.47, -16.5) mm, rotated rx -180 ry 0 rz 90 deg; joints [74.882, -18.394, 89.85, 0, 18.544, 74.882] to (-69.06, 50.96, -16.5) mm, rotated rx -180 ry 0 rz 90 deg; joints [74.864, -18.393, 89.846, 0, 18.547, 74.864]
  MoveL 9297 to (-69.06, 28.55, -16.5) mm, rotated rx -180 ry 0 rz 90 deg; joints [74.103, -18.302, 89.429, 0, 18.873, 74.103]
  MoveL 9298 to (-61.51, 28.55, -16.5) mm, rotated rx -180 ry 0 rz 90 deg; joints [74.175, -18.19, 88.921, 0, 19.268, 74.175]
  MoveL 9299 to (-61.51, 28.55, -13.5) mm, rotated rx -180 ry 0 rz 90 deg; joints [74.175, -18.347, 89.024, 0, 19.322, 74.175]
  Establecer velocidad (1000.0 mm/s)
  MoveL 9300 to (-61.51, 28.55, 10) mm, rotated rx 180 ry 0 rz 90 deg; joints [74.175, -19.574, 89.814, 0, 19.759, 74.175]
  Establecer velocidad (66.7 mm/s)
  MoveL 9301 to (-60.82, -44.42, 10) mm, rotated rx 180 ry 0 rz 90 deg; joints [71.754, -19.207, 88.257, 0, 20.95, 71.754]
  MoveL 9302 to (-60.82, -44.42, -13.25) mm, rotated rx 180 ry 0 rz 90 deg; joints [71.754, -18.001, 87.476, 0, 20.525, 71.754]
  MoveL 9303 to (-62.32, -44.23, -13.66) mm, rotated rx 180 ry 0 rz 90 deg; joints [71.743, -18.005, 87.568, 0, 20.437, 71.743]
  MoveL 9304 to (-63.83, -44.42, -14.06) mm, rotated rx 180 ry 0 rz 90 deg; joints [71.721, -18.007, 87.652, 0, 20.355, 71.721]
  MoveL 9305 to (-65.26, -44.93, -14.47) mm, rotated rx -180 ry 0 rz 90 deg; joints [71.689, -18.006, 87.723, 0, 20.283, 71.689]
  MoveL 9306 to (-66.55, -45.75, -14.87) mm, rotated rx 180 ry 0 rz 90 deg; joints [71.648, -18, 87.777, 0, 20.223, 71.648]
  MoveL 9307 to (-67.61, -46.82, -15.28) mm, rotated rx 180 ry 0 rz 90 deg; joints [71.6, -17.99, 87.811, 0, 20.179, 71.6]
  MoveL 9308 to (-68.42, -48.11, -15.69) mm, rotated rx 180 ry 0 rz 90 deg; joints [71.549, -17.975, 87.822, 0, 20.153, 71.549]
  MoveL 9309 to (-68.92, -49.55, -16.09) mm, rotated rx -180 ry 0 rz 90 deg; joints [71.496, -17.954, 87.81, 0, 20.145, 71.496]
  MoveL 9310 to (-69.06, -51.06, -16.5) mm, rotated rx 180 ry 0 rz 90 deg; joints [71.445, -17.927, 87.771, 0, 20.156, 71.445]
  MoveL 9311 to (-69.06, -65.86, -16.5) mm, rotated rx 180 ry 0 rz 90 deg; joints [70.96, -17.848, 87.432, 0, 20.416, 70.96]
  MoveL 9312 to (-69.04, -66.71, -16.5) mm, rotated rx -180 ry 0 rz 90 deg; joints [70.932, -17.843, 87.411, 0, 20.432, 70.932]
  MoveC 9313 to (-68.32, -68.34, -16.5) mm, rotated rx 180 ry 0 rz 90 deg; joints [70.887, -17.823, 87.325, 0, 20.498, 70.887] to (-66.66, -68.99, -16.5) mm, rotated rx 180 ry 0 rz 90 deg; joints [70.885, -17.793, 87.197, 0, 20.595, 70.885]
  MoveC 9314 to (-52.52, -68.66, -16.5) mm, rotated rx -180 ry 0 rz 90 deg; joints [71.054, -17.565, 86.246, 0, 21.319, 71.054] to (-38.38, -68.2, -16.5) mm, rotated rx 180 ry 0 rz 90 deg; joints [71.225, -17.328, 85.287, 0, 22.042, 71.225]
  MoveC 9315 to (-36.97, -67.62, -16.5) mm, rotated rx 180 ry 0 rz 90 deg; joints [71.259, -17.307, 85.203, 0, 22.104, 71.259] to (-36.16, -66.33, -16.5) mm, rotated rx 180 ry 0 rz 90 deg; joints [71.309, -17.301, 85.178, 0, 22.124, 71.309]
  MoveL 9316 to (-36.03, -65.86, -16.5) mm, rotated rx 180 ry 0 rz 90 deg; joints [71.326, -17.302, 85.18, 0, 22.122, 71.326]
  MoveL 9317 to (-26.93, -29.93, -16.5) mm, rotated rx 180 ry 0 rz 90 deg; joints [72.582, -17.347, 85.36, 0, 21.986, 72.582]
  MoveC 9318 to (-26.86, -29.2, -16.5) mm, rotated rx -180 ry 0 rz 90 deg; joints [72.607, -17.349, 85.371, 0, 21.978, 72.607] to (-27, -28.49, -16.5) mm, rotated rx 180 ry 0 rz 90 deg; joints [72.628, -17.356, 85.396, 0, 21.959, 72.628]
  MoveC 9319 to (-27.92, -27.12, -16.5) mm, rotated rx 180 ry 0 rz 90 deg; joints [72.664, -17.379, 85.49, 0, 21.889, 72.664] to (-29.36, -26.31, -16.5) mm, rotated rx 180 ry 0 rz 90 deg; joints [72.675, -17.408, 85.607, 0, 21.801, 72.675]
  MoveL 9320 to (-29.85, -26.37, -16.5) mm, rotated rx -180 ry 0 rz 90 deg; joints [72.669, -17.416, 85.64, 0, 21.776, 72.669]
  MoveL 9321 to (-30.04, -26.4, -16.5) mm, rotated rx 180 ry 0 rz 90 deg; joints [72.665, -17.419, 85.653, 0, 21.767, 72.665]
  MoveC 9322 to (-48.61, -29.87, -16.5) mm, rotated rx -180 ry 0 rz 90 deg; joints [72.361, -17.711, 86.855, 0, 20.857, 72.361] to (-67.16, -33.47, -16.5) mm, rotated rx -180 ry 0 rz 90 deg; joints [72.046, -17.988, 88.033, 0, 19.955, 72.046]
  MoveC 9323 to (-68.39, -34.15, -16.5) mm, rotated rx -180 ry 0 rz 90 deg; joints [72.01, -18.004, 88.102, 0, 19.902, 72.01] to (-69.01, -35.42, -16.5) mm, rotated rx 180 ry 0 rz 90 deg; joints [71.962, -18.007, 88.116, 0, 19.891, 71.962]
  MoveC 9324 to (-69.05, -35.69, -16.5) mm, rotated rx 180 ry 0 rz 90 deg; joints [71.952, -18.006, 88.112, 0, 19.894, 71.952] to (-69.06, -35.96, -16.5) mm, rotated rx -180 ry 0 rz 90 deg; joints [71.943, -18.005, 88.107, 0, 19.898, 71.943]
  MoveL 9325 to (-69.06, -51.06, -16.5) mm, rotated rx 180 ry 0 rz 90 deg; joints [71.445, -17.927, 87.771, 0, 20.156, 71.445]
  MoveL 9326 to (-61.51, -51.06, -16.5) mm, rotated rx -180 ry 0 rz 90 deg; joints [71.528, -17.808, 87.262, 0, 20.546, 71.528]
  MoveL 9327 to (-61.51, -51.06, -13.5) mm, rotated rx -180 ry 0 rz 90 deg; joints [71.528, -17.964, 87.365, 0, 20.599, 71.528]
  Establecer velocidad (1000.0 mm/s)
  MoveL 9328 to (-61.51, -51.06, 10) mm, rotated rx -180 ry 0 rz 90 deg; joints [71.528, -19.182, 88.154, 0, 21.028, 71.528]
  Establecer velocidad (66.7 mm/s)
  MoveL 9329 to (-60.65, -44.42, 10) mm, rotated rx 180 ry 0 rz 90 deg; joints [71.755, -19.204, 88.245, 0, 20.958, 71.755]
  MoveL 9330 to (-60.65, -44.42, -13.5) mm, rotated rx -180 ry 0 rz 90 deg; joints [71.755, -17.985, 87.456, 0, 20.529, 71.755]
  MoveL 9331 to (-62.16, -44.23, -13.91) mm, rotated rx 180 ry 0 rz 90 deg; joints [71.745, -17.989, 87.548, 0, 20.441, 71.745]
  MoveL 9332 to (-63.67, -44.42, -14.31) mm, rotated rx 180 ry 0 rz 90 deg; joints [71.723, -17.991, 87.632, 0, 20.359, 71.723]
  MoveL 9333 to (-65.1, -44.93, -14.72) mm, rotated rx 180 ry 0 rz 90 deg; joints [71.69, -17.99, 87.703, 0, 20.287, 71.69]
  MoveL 9334 to (-66.38, -45.75, -15.13) mm, rotated rx 180 ry 0 rz 90 deg; joints [71.65, -17.985, 87.757, 0, 20.227, 71.65]
  MoveL 9335 to (-67.45, -46.82, -15.53) mm, rotated rx 180 ry 0 rz 90 deg; joints [71.602, -17.975, 87.791, 0, 20.183, 71.602]
  MoveL 9336 to (-68.25, -48.11, -15.94) mm, rotated rx 180 ry 0 rz 90 deg; joints [71.551, -17.959, 87.803, 0, 20.157, 71.551]
  MoveL 9337 to (-68.75, -49.55, -16.34) mm, rotated rx 180 ry 0 rz 90 deg; joints [71.498, -17.939, 87.79, 0, 20.149, 71.498]
  MoveL 9338 to (-68.89, -51.06, -16.75) mm, rotated rx 180 ry 0 rz 90 deg; joints [71.447, -17.912, 87.751, 0, 20.161, 71.447]
  MoveL 9339 to (-68.89, -65.86, -16.75) mm, rotated rx -180 ry 0 rz 90 deg; joints [70.962, -17.833, 87.412, 0, 20.42, 70.962]
  MoveL 9340 to (-68.87, -66.59, -16.75) mm, rotated rx 180 ry 0 rz 90 deg; joints [70.938, -17.828, 87.394, 0, 20.434, 70.938]
  MoveC 9341 to (-68.18, -68.18, -16.75) mm, rotated rx -180 ry 0 rz 90 deg; joints [70.894, -17.809, 87.311, 0, 20.498, 70.894] to (-66.58, -68.84, -16.75) mm, rotated rx -180 ry 0 rz 90 deg; joints [70.89, -17.78, 87.187, 0, 20.593, 70.89]
  MoveC 9342 to (-64.8, -68.83, -16.75) mm, rotated rx 180 ry 0 rz 90 deg; joints [70.911, -17.751, 87.067, 0, 20.684, 70.911] to (-63.02, -68.77, -16.75) mm, rotated rx -180 ry 0 rz 90 deg; joints [70.933, -17.723, 86.948, 0, 20.775, 70.933]
  MoveC 9343 to (-50.79, -68.45, -16.75) mm, rotated rx 180 ry 0 rz 90 deg; joints [71.08, -17.524, 86.125, 0, 21.4, 71.08] to (-38.57, -68.04, -16.75) mm, rotated rx 180 ry 0 rz 90 deg; joints [71.228, -17.32, 85.295, 0, 22.024, 71.228]
  MoveC 9344 to (-37.11, -67.49, -16.75) mm, rotated rx 180 ry 0 rz 90 deg; joints [71.262, -17.298, 85.207, 0, 22.091, 71.262] to (-36.26, -66.17, -16.75) mm, rotated rx 180 ry 0 rz 90 deg; joints [71.313, -17.291, 85.18, 0, 22.111, 71.313]
  MoveL 9345 to (-27.07, -29.85, -16.75) mm, rotated rx 180 ry 0 rz 90 deg; joints [72.584, -17.337, 85.363, 0, 21.973, 72.584]
  MoveL 9346 to (-27.02, -29.56, -16.75) mm, rotated rx 180 ry 0 rz 90 deg; joints [72.593, -17.337, 85.366, 0, 21.972, 72.593]
  MoveC 9347 to (-27.64, -27.9, -16.75) mm, rotated rx -180 ry 0 rz 90 deg; joints [72.641, -17.357, 85.445, 0, 21.912, 72.641] to (-28.98, -26.72, -16.75) mm, rotated rx -180 ry 0 rz 90 deg; joints [72.666, -17.386, 85.563, 0, 21.823, 72.666]
  MoveC 9348 to (-29.46, -26.56, -16.75) mm, rotated rx -180 ry 0 rz 90 deg; joints [72.666, -17.396, 85.6, 0, 21.795, 72.666] to (-29.96, -26.57, -16.75) mm, rotated rx 180 ry 0 rz 90 deg; joints [72.661, -17.404, 85.635, 0, 21.769, 72.661]
  MoveC 9349 to (-48.5, -30.02, -16.75) mm, rotated rx 180 ry 0 rz 90 deg; joints [72.357, -17.696, 86.835, 0, 20.861, 72.357] to (-67, -33.59, -16.75) mm, rotated rx -180 ry 0 rz 90 deg; joints [72.044, -17.972, 88.012, 0, 19.96, 72.044]
  MoveC 9350 to (-68.25, -34.28, -16.75) mm, rotated rx 180 ry 0 rz 90 deg; joints [72.007, -17.988, 88.081, 0, 19.907, 72.007] to (-68.87, -35.58, -16.75) mm, rotated rx 180 ry 0 rz 90 deg; joints [71.958, -17.991, 88.094, 0, 19.897, 71.958]
  MoveC 9351 to (-68.89, -35.76, -16.75) mm, rotated rx 180 ry 0 rz 90 deg; joints [71.952, -17.99, 88.091, 0, 19.899, 71.952] to (-68.89, -35.95, -16.75) mm, rotated rx -180 ry 0 rz 90 deg; joints [71.945, -17.99, 88.087, 0, 19.902, 71.945]
  MoveL 9352 to (-68.89, -51.06, -16.75) mm, rotated rx 180 ry 0 rz 90 deg; joints [71.447, -17.912, 87.751, 0, 20.161, 71.447]
  MoveL 9353 to (-61.34, -51.06, -16.75) mm, rotated rx -180 ry 0 rz 90 deg; joints [71.53, -17.793, 87.242, 0, 20.551, 71.53]
  MoveL 9354 to (-61.34, -51.06, -13.75) mm, rotated rx 180 ry 0 rz 90 deg; joints [71.53, -17.948, 87.345, 0, 20.603, 71.53]
  Establecer velocidad (1000.0 mm/s)
  MoveL 9355 to (-61.34, -51.06, 10) mm, rotated rx 180 ry 0 rz 90 deg; joints [71.53, -19.179, 88.143, 0, 21.036, 71.53]
  Establecer velocidad (66.7 mm/s)
  MoveL 9356 to (-60.65, 35.1, 10) mm, rotated rx 180 ry 0 rz 90 deg; joints [74.404, -19.589, 89.881, 0, 19.708, 74.404]
  MoveL 9357 to (-60.65, 35.1, -13.5) mm, rotated rx 180 ry 0 rz 90 deg; joints [74.404, -18.362, 89.091, 0, 19.27, 74.404]
  MoveL 9358 to (-62.16, 35.29, -13.91) mm, rotated rx 180 ry 0 rz 90 deg; joints [74.396, -18.364, 89.182, 0, 19.181, 74.396]
  MoveL 9359 to (-63.67, 35.11, -14.31) mm, rotated rx -180 ry 0 rz 90 deg; joints [74.376, -18.364, 89.266, 0, 19.098, 74.376]
  MoveL 9360 to (-65.1, 34.59, -14.72) mm, rotated rx 180 ry 0 rz 90 deg; joints [74.345, -18.362, 89.339, 0, 19.023, 74.345]
  MoveL 9361 to (-66.38, 33.78, -15.13) mm, rotated rx -180 ry 0 rz 90 deg; joints [74.305, -18.357, 89.396, 0, 18.961, 74.305]
  MoveL 9362 to (-67.45, 32.7, -15.53) mm, rotated rx -180 ry 0 rz 90 deg; joints [74.259, -18.347, 89.433, 0, 18.913, 74.259]
  MoveL 9363 to (-68.25, 31.41, -15.94) mm, rotated rx 180 ry 0 rz 90 deg; joints [74.207, -18.332, 89.449, 0, 18.883, 74.207]
  MoveL 9364 to (-68.75, 29.97, -16.34) mm, rotated rx 180 ry 0 rz 90 deg; joints [74.154, -18.312, 89.441, 0, 18.871, 74.154]
  MoveL 9365 to (-68.89, 28.46, -16.75) mm, rotated rx -180 ry 0 rz 90 deg; joints [74.101, -18.287, 89.408, 0, 18.879, 74.101]
  MoveL 9366 to (-68.89, 6.16, -16.75) mm, rotated rx -180 ry 0 rz 90 deg; joints [73.349, -18.19, 88.971, 0, 19.219, 73.349]
  MoveC 9367 to (-67.93, 4.28, -16.75) mm, rotated rx -180 ry 0 rz 90 deg; joints [73.296, -18.167, 88.869, 0, 19.298, 73.296] to (-65.86, 3.86, -16.75) mm, rotated rx -180 ry 0 rz 90 deg; joints [73.303, -18.134, 88.721, 0, 19.412, 73.303]
  MoveC 9368 to (-46.65, 8.65, -16.75) mm, rotated rx 180 ry 0 rz 90 deg; joints [73.653, -17.857, 87.516, 0, 20.341, 73.653] to (-27.48, 13.61, -16.75) mm, rotated rx 180 ry 0 rz 90 deg; joints [74.001, -17.566, 86.297, 0, 21.269, 74.001]
  MoveC 9369 to (-26.17, 14.83, -16.75) mm, rotated rx 180 ry 0 rz 90 deg; joints [74.053, -17.55, 86.23, 0, 21.32, 74.053] to (-25.86, 16.58, -16.75) mm, rotated rx 180 ry 0 rz 90 deg; joints [74.114, -17.553, 86.243, 0, 21.31, 74.114]
  MoveL 9370 to (-26.06, 17.26, -16.75) mm, rotated rx -180 ry 0 rz 90 deg; joints [74.134, -17.56, 86.271, 0, 21.289, 74.134]
  MoveL 9371 to (-29.98, 28.53, -16.75) mm, rotated rx 180 ry 0 rz 90 deg; joints [74.47, -17.678, 86.761, 0, 20.917, 74.47]
  MoveC 9372 to (-30.37, 29.26, -16.75) mm, rotated rx 180 ry 0 rz 90 deg; joints [74.491, -17.688, 86.802, 0, 20.886, 74.491] to (-30.97, 29.83, -16.75) mm, rotated rx -180 ry 0 rz 90 deg; joints [74.504, -17.701, 86.854, 0, 20.846, 74.504]
  MoveC 9373 to (-48.15, 41.39, -16.75) mm, rotated rx -180 ry 0 rz 90 deg; joints [74.733, -18.027, 88.25, 0, 19.777, 74.733] to (-65.41, 52.82, -16.75) mm, rotated rx -180 ry 0 rz 90 deg; joints [74.961, -18.334, 89.626, 0, 18.708, 74.961]
  MoveC 9374 to (-67.19, 52.71, -16.75) mm, rotated rx -180 ry 0 rz 90 deg; joints [74.941, -18.36, 89.744, 0, 18.616, 74.941] to (-68.61, 51.63, -16.75) mm, rotated rx 180 ry 0 rz 90 deg; joints [74.891, -18.376, 89.82, 0, 18.557, 74.891]
  MoveC 9375 to (-68.82, 51.22, -16.75) mm, rotated rx 180 ry 0 rz 90 deg; joints [74.875, -18.378, 89.826, 0, 18.551, 74.875] to (-68.89, 50.77, -16.75) mm, rotated rx -180 ry 0 rz 90 deg; joints [74.859, -18.377, 89.823, 0, 18.554, 74.859]
  MoveL 9376 to (-68.89, 28.46, -16.75) mm, rotated rx -180 ry 0 rz 90 deg; joints [74.101, -18.287, 89.408, 0, 18.879, 74.101]
  MoveL 9377 to (-61.34, 28.46, -16.75) mm, rotated rx 180 ry 0 rz 90 deg; joints [74.174, -18.174, 88.9, 0, 19.274, 74.174]
  MoveL 9378 to (-61.34, 28.46, -13.75) mm, rotated rx 180 ry 0 rz 90 deg; joints [74.174, -18.331, 89.003, 0, 19.328, 74.174]
  Establecer velocidad (1000.0 mm/s)
  MoveL 9379 to (-61.34, 28.46, 10) mm, rotated rx -180 ry 0 rz 90 deg; joints [74.174, -19.571, 89.802, 0, 19.769, 74.174]
  Establecer velocidad (66.7 mm/s)
  MoveL 9380 to (-60.49, 35.1, 10) mm, rotated rx 180 ry 0 rz 90 deg; joints [74.406, -19.587, 89.87, 0, 19.717, 74.406]
  MoveL 9381 to (-60.49, 35.1, -13.75) mm, rotated rx 180 ry 0 rz 90 deg; joints [74.406, -18.346, 89.072, 0, 19.274, 74.406]
  MoveL 9382 to (-61.99, 35.29, -14.16) mm, rotated rx 180 ry 0 rz 90 deg; joints [74.398, -18.348, 89.163, 0, 19.186, 74.398]
  MoveL 9383 to (-63.5, 35.11, -14.56) mm, rotated rx 180 ry 0 rz 90 deg; joints [74.378, -18.349, 89.247, 0, 19.102, 74.378]
  MoveL 9384 to (-64.93, 34.59, -14.97) mm, rotated rx 180 ry 0 rz 90 deg; joints [74.347, -18.347, 89.319, 0, 19.027, 74.347]
  MoveL 9385 to (-66.22, 33.78, -15.37) mm, rotated rx 180 ry 0 rz 90 deg; joints [74.307, -18.341, 89.376, 0, 18.965, 74.307]
  MoveL 9386 to (-67.28, 32.7, -15.78) mm, rotated rx 180 ry 0 rz 90 deg; joints [74.26, -18.331, 89.414, 0, 18.917, 74.26]
  MoveL 9387 to (-68.09, 31.41, -16.19) mm, rotated rx -180 ry 0 rz 90 deg; joints [74.209, -18.316, 89.429, 0, 18.887, 74.209]
  MoveL 9388 to (-68.59, 29.97, -16.59) mm, rotated rx -180 ry 0 rz 90 deg; joints [74.155, -18.297, 89.422, 0, 18.875, 74.155]
  MoveL 9389 to (-68.73, 28.46, -17) mm, rotated rx 180 ry 0 rz 90 deg; joints [74.103, -18.271, 89.388, 0, 18.883, 74.103]
  MoveL 9390 to (-68.73, 7.11, -17) mm, rotated rx 180 ry 0 rz 90 deg; joints [73.383, -18.178, 88.97, 0, 19.208, 73.383]
  MoveL 9391 to (-68.72, 6.16, -17) mm, rotated rx 180 ry 0 rz 90 deg; joints [73.351, -18.174, 88.951, 0, 19.223, 73.351]
  MoveC 9392 to (-67.77, 4.45, -17) mm, rotated rx -180 ry 0 rz 90 deg; joints [73.303, -18.152, 88.853, 0, 19.299, 73.303] to (-65.86, 4.01, -17) mm, rotated rx -180 ry 0 rz 90 deg; joints [73.308, -18.121, 88.716, 0, 19.406, 73.308]
  MoveC 9393 to (-46.74, 8.79, -17) mm, rotated rx -180 ry 0 rz 90 deg; joints [73.656, -17.846, 87.516, 0, 20.33, 73.656] to (-27.67, 13.74, -17) mm, rotated rx 180 ry 0 rz 90 deg; joints [74.003, -17.557, 86.304, 0, 21.253, 74.003]
  MoveC 9394 to (-26.38, 14.95, -17) mm, rotated rx 180 ry 0 rz 90 deg; joints [74.055, -17.541, 86.238, 0, 21.303, 74.055] to (-26.06, 16.68, -17) mm, rotated rx -180 ry 0 rz 90 deg; joints [74.115, -17.544, 86.25, 0, 21.294, 74.115]
  MoveL 9395 to (-26.32, 17.53, -17) mm, rotated rx -180 ry 0 rz 90 deg; joints [74.141, -17.553, 86.285, 0, 21.267, 74.141]
  MoveL 9396 to (-29.28, 26.06, -17) mm, rotated rx -180 ry 0 rz 90 deg; joints [74.395, -17.642, 86.656, 0, 20.986, 74.395]
  MoveL 9397 to (-29.6, 27.01, -17) mm, rotated rx 180 ry 0 rz 90 deg; joints [74.423, -17.652, 86.697, 0, 20.955, 74.423]
  MoveC 9398 to (-29.9, 27.85, -17) mm, rotated rx -180 ry 0 rz 90 deg; joints [74.449, -17.661, 86.733, 0, 20.927, 74.449] to (-30.22, 28.68, -17) mm, rotated rx -180 ry 0 rz 90 deg; joints [74.473, -17.67, 86.772, 0, 20.898, 74.473]
  MoveC 9399 to (-30.56, 29.25, -17) mm, rotated rx 180 ry 0 rz 90 deg; joints [74.489, -17.678, 86.806, 0, 20.872, 74.489] to (-31.05, 29.69, -17) mm, rotated rx -180 ry 0 rz 90 deg; joints [74.499, -17.688, 86.848, 0, 20.84, 74.499]
  MoveC 9400 to (-48.12, 41.19, -17) mm, rotated rx 180 ry 0 rz 90 deg; joints [74.726, -18.012, 88.235, 0, 19.777, 74.726] to (-65.26, 52.58, -17) mm, rotated rx -180 ry 0 rz 90 deg; joints [74.954, -18.318, 89.604, 0, 18.715, 74.954]
  MoveC 9401 to (-67.16, 52.42, -17) mm, rotated rx 180 ry 0 rz 90 deg; joints [74.932, -18.345, 89.728, 0, 18.617, 74.932] to (-68.59, 51.17, -17) mm, rotated rx 180 ry 0 rz 90 deg; joints [74.876, -18.361, 89.801, 0, 18.56, 74.876]
  MoveC 9402 to (-68.69, 50.95, -17) mm, rotated rx 180 ry 0 rz 90 deg; joints [74.867, -18.362, 89.804, 0, 18.558, 74.867] to (-68.73, 50.7, -17) mm, rotated rx -180 ry 0 rz 90 deg; joints [74.858, -18.361, 89.802, 0, 18.559, 74.858]
  MoveL 9403 to (-68.73, 28.46, -17) mm, rotated rx 180 ry 0 rz 90 deg; joints [74.103, -18.271, 89.388, 0, 18.883, 74.103]
  MoveL 9404 to (-61.18, 28.46, -17) mm, rotated rx -180 ry 0 rz 90 deg; joints [74.175, -18.158, 88.881, 0, 19.278, 74.175]
  MoveL 9405 to (-61.18, 28.46, -14) mm, rotated rx -180 ry 0 rz 90 deg; joints [74.175, -18.315, 88.984, 0, 19.332, 74.175]
  Establecer velocidad (1000.0 mm/s)
  MoveL 9406 to (-61.18, 28.46, 10) mm, rotated rx -180 ry 0 rz 90 deg; joints [74.175, -19.568, 89.791, 0, 19.778, 74.175]
  Establecer velocidad (66.7 mm/s)
  MoveL 9407 to (-60.49, -44.37, 10) mm, rotated rx 180 ry 0 rz 90 deg; joints [71.759, -19.201, 88.235, 0, 20.966, 71.759]
  MoveL 9408 to (-60.49, -44.37, -13.75) mm, rotated rx -180 ry 0 rz 90 deg; joints [71.759, -17.97, 87.437, 0, 20.533, 71.759]
  MoveL 9409 to (-61.99, -44.18, -14.16) mm, rotated rx 180 ry 0 rz 90 deg; joints [71.749, -17.974, 87.529, 0, 20.445, 71.749]
  MoveL 9410 to (-63.5, -44.37, -14.56) mm, rotated rx 180 ry 0 rz 90 deg; joints [71.726, -17.976, 87.613, 0, 20.362, 71.726]
  MoveL 9411 to (-64.93, -44.88, -14.97) mm, rotated rx 180 ry 0 rz 90 deg; joints [71.694, -17.975, 87.685, 0, 20.29, 71.694]
  MoveL 9412 to (-66.22, -45.69, -15.37) mm, rotated rx 180 ry 0 rz 90 deg; joints [71.653, -17.969, 87.739, 0, 20.231, 71.653]
  MoveL 9413 to (-67.28, -46.77, -15.78) mm, rotated rx 180 ry 0 rz 90 deg; joints [71.606, -17.959, 87.773, 0, 20.187, 71.606]
  MoveL 9414 to (-68.09, -48.06, -16.19) mm, rotated rx 180 ry 0 rz 90 deg; joints [71.555, -17.944, 87.784, 0, 20.16, 71.555]
  MoveL 9415 to (-68.59, -49.5, -16.59) mm, rotated rx -180 ry 0 rz 90 deg; joints [71.502, -17.923, 87.772, 0, 20.152, 71.502]
  MoveL 9416 to (-68.73, -51.01, -17) mm, rotated rx -180 ry 0 rz 90 deg; joints [71.451, -17.896, 87.733, 0, 20.164, 71.451]
  MoveL 9417 to (-68.73, -65.86, -17) mm, rotated rx 180 ry 0 rz 90 deg; joints [70.964, -17.817, 87.393, 0, 20.424, 70.964]
  MoveL 9418 to (-68.71, -66.48, -17) mm, rotated rx 180 ry 0 rz 90 deg; joints [70.943, -17.813, 87.377, 0, 20.436, 70.943]
  MoveC 9419 to (-68.01, -68.07, -17) mm, rotated rx -180 ry 0 rz 90 deg; joints [70.9, -17.793, 87.293, 0, 20.501, 70.9] to (-66.39, -68.7, -17) mm, rotated rx 180 ry 0 rz 90 deg; joints [70.897, -17.764, 87.169, 0, 20.596, 70.897]
  MoveC 9420 to (-53.64, -68.38, -17) mm, rotated rx -180 ry 0 rz 90 deg; joints [71.05, -17.559, 86.312, 0, 21.247, 71.05] to (-40.9, -67.96, -17) mm, rotated rx -180 ry 0 rz 90 deg; joints [71.205, -17.347, 85.449, 0, 21.898, 71.205]
  MoveC 9421 to (-39.64, -67.91, -17) mm, rotated rx 180 ry 0 rz 90 deg; joints [71.22, -17.326, 85.363, 0, 21.963, 71.22] to (-38.38, -67.86, -17) mm, rotated rx -180 ry 0 rz 90 deg; joints [71.236, -17.305, 85.278, 0, 22.027, 71.236]
  MoveC 9422 to (-37.23, -67.35, -17) mm, rotated rx 180 ry 0 rz 90 deg; joints [71.265, -17.288, 85.21, 0, 22.077, 71.265] to (-36.48, -66.34, -17) mm, rotated rx -180 ry 0 rz 90 deg; joints [71.305, -17.281, 85.182, 0, 22.098, 71.305]
  MoveL 9423 to (-36.34, -65.86, -17) mm, rotated rx -180 ry 0 rz 90 deg; joints [71.322, -17.281, 85.183, 0, 22.098, 71.322]
  MoveL 9424 to (-27.24, -29.85, -17) mm, rotated rx 180 ry 0 rz 90 deg; joints [72.582, -17.327, 85.366, 0, 21.961, 72.582]
  MoveC 9425 to (-28.02, -27.85, -17) mm, rotated rx 180 ry 0 rz 90 deg; joints [72.639, -17.351, 85.464, 0, 21.887, 72.639] to (-29.85, -26.73, -17) mm, rotated rx 180 ry 0 rz 90 deg; joints [72.657, -17.388, 85.615, 0, 21.773, 72.657]
  MoveC 9426 to (-48.34, -30.15, -17) mm, rotated rx 180 ry 0 rz 90 deg; joints [72.355, -17.68, 86.813, 0, 20.867, 72.355] to (-66.81, -33.71, -17) mm, rotated rx 180 ry 0 rz 90 deg; joints [72.042, -17.955, 87.988, 0, 19.968, 72.042]
  MoveC 9427 to (-68.03, -34.33, -17) mm, rotated rx -180 ry 0 rz 90 deg; joints [72.008, -17.971, 88.056, 0, 19.915, 72.008] to (-68.69, -35.54, -17) mm, rotated rx 180 ry 0 rz 90 deg; joints [71.961, -17.975, 88.074, 0, 19.901, 71.961]
  MoveL 9428 to (-68.7, -35.73, -17) mm, rotated rx 180 ry 0 rz 90 deg; joints [71.955, -17.975, 88.071, 0, 19.904, 71.955]
  MoveL 9429 to (-68.73, -36.48, -17) mm, rotated rx -180 ry 0 rz 90 deg; joints [71.93, -17.971, 88.056, 0, 19.915, 71.93]
  MoveL 9430 to (-68.73, -51.01, -17) mm, rotated rx -180 ry 0 rz 90 deg; joints [71.451, -17.896, 87.733, 0, 20.164, 71.451]
  MoveL 9431 to (-61.18, -51.01, -17) mm, rotated rx -180 ry 0 rz 90 deg; joints [71.534, -17.777, 87.223, 0, 20.554, 71.534]
  MoveL 9432 to (-61.18, -51.01, -14) mm, rotated rx 180 ry 0 rz 90 deg; joints [71.534, -17.933, 87.326, 0, 20.606, 71.534]
  Establecer velocidad (1000.0 mm/s)
  MoveL 9433 to (-61.18, -51.01, 10) mm, rotated rx 180 ry 0 rz 90 deg; joints [71.534, -19.177, 88.133, 0, 21.044, 71.534]
  Establecer velocidad (66.7 mm/s)
  MoveL 9434 to (-60.32, -44.37, 10) mm, rotated rx 180 ry 0 rz 90 deg; joints [71.761, -19.199, 88.224, 0, 20.974, 71.761]
  MoveL 9435 to (-60.32, -44.37, -14) mm, rotated rx 180 ry 0 rz 90 deg; joints [71.761, -17.954, 87.418, 0, 20.537, 71.761]
  MoveL 9436 to (-61.83, -44.18, -14.41) mm, rotated rx -180 ry 0 rz 90 deg; joints [71.75, -17.958, 87.51, 0, 20.449, 71.75]
  MoveL 9437 to (-63.34, -44.37, -14.81) mm, rotated rx 180 ry 0 rz 90 deg; joints [71.728, -17.96, 87.594, 0, 20.367, 71.728]
  MoveL 9438 to (-64.77, -44.88, -15.22) mm, rotated rx 180 ry 0 rz 90 deg; joints [71.696, -17.959, 87.665, 0, 20.294, 71.696]
  MoveL 9439 to (-66.05, -45.69, -15.63) mm, rotated rx -180 ry 0 rz 90 deg; joints [71.655, -17.954, 87.719, 0, 20.235, 71.655]
  MoveL 9440 to (-67.12, -46.77, -16.03) mm, rotated rx -180 ry 0 rz 90 deg; joints [71.608, -17.944, 87.753, 0, 20.191, 71.608]
  MoveL 9441 to (-67.92, -48.06, -16.44) mm, rotated rx -180 ry 0 rz 90 deg; joints [71.556, -17.929, 87.764, 0, 20.164, 71.556]
  MoveL 9442 to (-68.42, -49.5, -16.84) mm, rotated rx -180 ry 0 rz 90 deg; joints [71.504, -17.908, 87.752, 0, 20.156, 71.504]
  MoveL 9443 to (-68.56, -51.01, -17.25) mm, rotated rx -180 ry 0 rz 90 deg; joints [71.452, -17.881, 87.713, 0, 20.168, 71.452]
  MoveL 9444 to (-68.56, -65.86, -17.25) mm, rotated rx 180 ry 0 rz 90 deg; joints [70.965, -17.801, 87.373, 0, 20.429, 70.965]
  MoveL 9445 to (-68.56, -66.28, -17.25) mm, rotated rx -180 ry 0 rz 90 deg; joints [70.952, -17.799, 87.363, 0, 20.436, 70.952]
  MoveC 9446 to (-67.85, -67.91, -17.25) mm, rotated rx -180 ry 0 rz 90 deg; joints [70.906, -17.779, 87.277, 0, 20.502, 70.906] to (-66.2, -68.56, -17.25) mm, rotated rx -180 ry 0 rz 90 deg; joints [70.904, -17.749, 87.151, 0, 20.598, 70.904]
  MoveC 9447 to (-53.34, -68.22, -17.25) mm, rotated rx 180 ry 0 rz 90 deg; joints [71.059, -17.542, 86.287, 0, 21.255, 71.059] to (-40.48, -67.78, -17.25) mm, rotated rx -180 ry 0 rz 90 deg; joints [71.215, -17.328, 85.416, 0, 21.913, 71.215]
  MoveC 9448 to (-39.59, -67.75, -17.25) mm, rotated rx 180 ry 0 rz 90 deg; joints [71.226, -17.313, 85.355, 0, 21.958, 71.226] to (-38.7, -67.71, -17.25) mm, rotated rx -180 ry 0 rz 90 deg; joints [71.237, -17.298, 85.295, 0, 22.003, 71.237]
  MoveC 9449 to (-37.3, -67.16, -17.25) mm, rotated rx -180 ry 0 rz 90 deg; joints [71.27, -17.277, 85.211, 0, 22.066, 71.27] to (-36.5, -65.9, -17.25) mm, rotated rx 180 ry 0 rz 90 deg; joints [71.319, -17.271, 85.185, 0, 22.086, 71.319]
  MoveL 9450 to (-28.9, -35.83, -17.25) mm, rotated rx -180 ry 0 rz 90 deg; joints [72.371, -17.31, 85.342, 0, 21.968, 72.371]
  MoveL 9451 to (-27.64, -30.8, -17.25) mm, rotated rx -180 ry 0 rz 90 deg; joints [72.547, -17.316, 85.365, 0, 21.951, 72.547]
  MoveL 9452 to (-27.44, -29.85, -17.25) mm, rotated rx 180 ry 0 rz 90 deg; joints [72.58, -17.317, 85.372, 0, 21.946, 72.58]
  MoveC 9453 to (-28.27, -28.02, -17.25) mm, rotated rx 180 ry 0 rz 90 deg; joints [72.631, -17.342, 85.469, 0, 21.872, 72.631] to (-29.97, -26.95, -17.25) mm, rotated rx 180 ry 0 rz 90 deg; joints [72.648, -17.376, 85.61, 0, 21.766, 72.648]
  MoveC 9454 to (-48.41, -30.32, -17.25) mm, rotated rx 180 ry 0 rz 90 deg; joints [72.348, -17.667, 86.805, 0, 20.862, 72.348] to (-66.81, -33.86, -17.25) mm, rotated rx 180 ry 0 rz 90 deg; joints [72.037, -17.942, 87.976, 0, 19.966, 72.037]
  MoveC 9455 to (-68.05, -34.64, -17.25) mm, rotated rx -180 ry 0 rz 90 deg; joints [71.998, -17.957, 88.042, 0, 19.915, 71.998] to (-68.55, -36.01, -17.25) mm, rotated rx 180 ry 0 rz 90 deg; joints [71.947, -17.958, 88.046, 0, 19.912, 71.947]
  MoveL 9456 to (-68.56, -36.48, -17.25) mm, rotated rx -180 ry 0 rz 90 deg; joints [71.931, -17.956, 88.036, 0, 19.919, 71.931]
  MoveL 9457 to (-68.56, -51.01, -17.25) mm, rotated rx -180 ry 0 rz 90 deg; joints [71.452, -17.881, 87.713, 0, 20.168, 71.452]
  MoveL 9458 to (-61.01, -51.01, -17.25) mm, rotated rx -180 ry 0 rz 90 deg; joints [71.535, -17.762, 87.204, 0, 20.558, 71.535]
  MoveL 9459 to (-61.01, -51.01, -14.25) mm, rotated rx 180 ry 0 rz 90 deg; joints [71.535, -17.917, 87.307, 0, 20.611, 71.535]
  Establecer velocidad (1000.0 mm/s)
  MoveL 9460 to (-61.01, -51.01, 10) mm, rotated rx 180 ry 0 rz 90 deg; joints [71.535, -19.174, 88.122, 0, 21.052, 71.535]
  Establecer velocidad (66.7 mm/s)
  MoveL 9461 to (-60.33, 35.12, 10) mm, rotated rx 180 ry 0 rz 90 deg; joints [74.408, -19.584, 89.859, 0, 19.725, 74.408]
  MoveL 9462 to (-60.32, 35.12, -14) mm, rotated rx 180 ry 0 rz 90 deg; joints [74.408, -18.331, 89.052, 0, 19.278, 74.408]
  MoveL 9463 to (-61.83, 35.3, -14.41) mm, rotated rx 180 ry 0 rz 90 deg; joints [74.4, -18.333, 89.143, 0, 19.19, 74.4]
  MoveL 9464 to (-63.34, 35.12, -14.81) mm, rotated rx 180 ry 0 rz 90 deg; joints [74.38, -18.333, 89.227, 0, 19.106, 74.38]
  MoveL 9465 to (-64.77, 34.61, -15.22) mm, rotated rx -180 ry 0 rz 90 deg; joints [74.349, -18.331, 89.3, 0, 19.031, 74.349]
  MoveL 9466 to (-66.05, 33.79, -15.63) mm, rotated rx -180 ry 0 rz 90 deg; joints [74.309, -18.326, 89.357, 0, 18.969, 74.309]
  MoveL 9467 to (-67.12, 32.71, -16.03) mm, rotated rx 180 ry 0 rz 90 deg; joints [74.262, -18.316, 89.394, 0, 18.921, 74.262]
  MoveL 9468 to (-67.92, 31.42, -16.44) mm, rotated rx 180 ry 0 rz 90 deg; joints [74.211, -18.301, 89.41, 0, 18.891, 74.211]
  MoveL 9469 to (-68.43, 29.99, -16.84) mm, rotated rx 180 ry 0 rz 90 deg; joints [74.157, -18.281, 89.402, 0, 18.879, 74.157]
  MoveL 9470 to (-68.56, 28.48, -17.25) mm, rotated rx -180 ry 0 rz 90 deg; joints [74.105, -18.256, 89.369, 0, 18.887, 74.105]
  MoveL 9471 to (-68.56, 6.63, -17.25) mm, rotated rx 180 ry 0 rz 90 deg; joints [73.369, -18.161, 88.941, 0, 19.219, 73.369]
  MoveC 9472 to (-67.79, 4.77, -17.25) mm, rotated rx 180 ry 0 rz 90 deg; joints [73.314, -18.141, 88.852, 0, 19.289, 73.314] to (-65.86, 4.16, -17.25) mm, rotated rx 180 ry 0 rz 90 deg; joints [73.313, -18.109, 88.71, 0, 19.399, 73.313]
  MoveL 9473 to (-65.39, 4.26, -17.25) mm, rotated rx 180 ry 0 rz 90 deg; joints [73.321, -18.102, 88.68, 0, 19.422, 73.321]
  MoveC 9474 to (-46.69, 8.96, -17.25) mm, rotated rx -180 ry 0 rz 90 deg; joints [73.662, -17.833, 87.508, 0, 20.325, 73.662] to (-28.03, 13.8, -17.25) mm, rotated rx -180 ry 0 rz 90 deg; joints [74.002, -17.551, 86.322, 0, 21.229, 74.002]
  MoveC 9475 to (-27.72, 13.92, -17.25) mm, rotated rx -180 ry 0 rz 90 deg; joints [74.009, -17.546, 86.302, 0, 21.244, 74.009] to (-27.43, 14.09, -17.25) mm, rotated rx -180 ry 0 rz 90 deg; joints [74.017, -17.542, 86.285, 0, 21.257, 74.017]
  MoveC 9476 to (-26.52, 15.19, -17.25) mm, rotated rx -180 ry 0 rz 90 deg; joints [74.062, -17.532, 86.244, 0, 21.288, 74.062] to (-26.23, 16.58, -17.25) mm, rotated rx -180 ry 0 rz 90 deg; joints [74.11, -17.534, 86.251, 0, 21.282, 74.11]
  MoveL 9477 to (-26.49, 17.53, -17.25) mm, rotated rx 180 ry 0 rz 90 deg; joints [74.139, -17.543, 86.288, 0, 21.254, 74.139]
  MoveL 9478 to (-27.01, 19.02, -17.25) mm, rotated rx 180 ry 0 rz 90 deg; joints [74.183, -17.558, 86.353, 0, 21.205, 74.183]
  MoveL 9479 to (-29.96, 27.57, -17.25) mm, rotated rx -180 ry 0 rz 90 deg; joints [74.439, -17.647, 86.724, 0, 20.924, 74.439]
  MoveC 9480 to (-30.21, 28.24, -17.25) mm, rotated rx -180 ry 0 rz 90 deg; joints [74.459, -17.655, 86.754, 0, 20.9, 74.459] to (-30.51, 28.9, -17.25) mm, rotated rx -180 ry 0 rz 90 deg; joints [74.478, -17.663, 86.788, 0, 20.875, 74.478]
  MoveC 9481 to (-30.87, 29.33, -17.25) mm, rotated rx 180 ry 0 rz 90 deg; joints [74.488, -17.671, 86.821, 0, 20.85, 74.488] to (-31.31, 29.68, -17.25) mm, rotated rx 180 ry 0 rz 90 deg; joints [74.496, -17.679, 86.857, 0, 20.822, 74.496]
  MoveC 9482 to (-48.18, 41.06, -17.25) mm, rotated rx 180 ry 0 rz 90 deg; joints [74.721, -18, 88.229, 0, 19.771, 74.721] to (-65.13, 52.33, -17.25) mm, rotated rx 180 ry 0 rz 90 deg; joints [74.947, -18.302, 89.582, 0, 18.72, 74.947]
  MoveC 9483 to (-66.88, 52.22, -17.25) mm, rotated rx -180 ry 0 rz 90 deg; joints [74.927, -18.327, 89.697, 0, 18.63, 74.927] to (-68.29, 51.17, -17.25) mm, rotated rx -180 ry 0 rz 90 deg; joints [74.879, -18.344, 89.773, 0, 18.571, 74.879]
  MoveC 9484 to (-68.51, 50.77, -17.25) mm, rotated rx 180 ry 0 rz 90 deg; joints [74.863, -18.345, 89.78, 0, 18.565, 74.863] to (-68.56, 50.32, -17.25) mm, rotated rx 180 ry 0 rz 90 deg; joints [74.847, -18.344, 89.776, 0, 18.569, 74.847]
  MoveL 9485 to (-68.56, 28.48, -17.25) mm, rotated rx -180 ry 0 rz 90 deg; joints [74.105, -18.256, 89.369, 0, 18.887, 74.105]
  MoveL 9486 to (-61.01, 28.48, -17.25) mm, rotated rx -180 ry 0 rz 90 deg; joints [74.177, -18.143, 88.861, 0, 19.282, 74.177]
  MoveL 9487 to (-61.01, 28.48, -14.25) mm, rotated rx 180 ry 0 rz 90 deg; joints [74.177, -18.3, 88.964, 0, 19.336, 74.177]
  Establecer velocidad (1000.0 mm/s)
  MoveL 9488 to (-61.01, 28.48, 10) mm, rotated rx -180 ry 0 rz 90 deg; joints [74.177, -19.566, 89.78, 0, 19.786, 74.177]
  Establecer velocidad (66.7 mm/s)
  MoveL 9489 to (-60.16, 35.12, 10) mm, rotated rx -180 ry 0 rz 90 deg; joints [74.41, -19.582, 89.848, 0, 19.733, 74.41]
  MoveL 9490 to (-60.16, 35.12, -14.25) mm, rotated rx -180 ry 0 rz 90 deg; joints [74.41, -18.315, 89.033, 0, 19.282, 74.41]
  MoveL 9491 to (-61.67, 35.3, -14.66) mm, rotated rx 180 ry 0 rz 90 deg; joints [74.402, -18.317, 89.124, 0, 19.194, 74.402]
  MoveL 9492 to (-63.17, 35.12, -15.06) mm, rotated rx -180 ry 0 rz 90 deg; joints [74.381, -18.318, 89.208, 0, 19.11, 74.381]
  MoveL 9493 to (-64.6, 34.61, -15.47) mm, rotated rx 180 ry 0 rz 90 deg; joints [74.35, -18.316, 89.281, 0, 19.035, 74.35]
  MoveL 9494 to (-65.89, 33.79, -15.87) mm, rotated rx -180 ry 0 rz 90 deg; joints [74.311, -18.31, 89.337, 0, 18.973, 74.311]
  MoveL 9495 to (-66.96, 32.71, -16.28) mm, rotated rx -180 ry 0 rz 90 deg; joints [74.264, -18.3, 89.375, 0, 18.925, 74.264]
  MoveL 9496 to (-67.76, 31.42, -16.69) mm, rotated rx -180 ry 0 rz 90 deg; joints [74.212, -18.285, 89.39, 0, 18.895, 74.212]
  MoveL 9497 to (-68.26, 29.99, -17.09) mm, rotated rx 180 ry 0 rz 90 deg; joints [74.159, -18.265, 89.383, 0, 18.883, 74.159]
  MoveL 9498 to (-68.4, 28.48, -17.5) mm, rotated rx -180 ry 0 rz 90 deg; joints [74.107, -18.24, 89.349, 0, 18.891, 74.107]
  MoveL 9499 to (-68.4, 6.63, -17.5) mm, rotated rx 180 ry 0 rz 90 deg; joints [73.37, -18.145, 88.922, 0, 19.224, 73.37]
  MoveC 9500 to (-67.45, 4.78, -17.5) mm, rotated rx -180 ry 0 rz 90 deg; joints [73.317, -18.122, 88.82, 0, 19.302, 73.317] to (-65.39, 4.41, -17.5) mm, rotated rx 180 ry 0 rz 90 deg; joints [73.326, -18.09, 88.675, 0, 19.415, 73.326]
  MoveC 9501 to (-47.13, 9.01, -17.5) mm, rotated rx 180 ry 0 rz 90 deg; joints [73.66, -17.827, 87.53, 0, 20.297, 73.66] to (-28.91, 13.75, -17.5) mm, rotated rx 180 ry 0 rz 90 deg; joints [73.992, -17.552, 86.372, 0, 21.18, 73.992]
  MoveL 9502 to (-28.91, 24, -17.5) mm, rotated rx 180 ry 0 rz 90 deg; joints [74.33, -17.6, 86.573, 0, 21.027, 74.33]
  MoveL 9503 to (-30.08, 27.46, -17.5) mm, rotated rx 180 ry 0 rz 90 deg; joints [74.434, -17.636, 86.721, 0, 20.915, 74.434]
  MoveC 9504 to (-30.36, 28.19, -17.5) mm, rotated rx -180 ry 0 rz 90 deg; joints [74.456, -17.644, 86.755, 0, 20.889, 74.456] to (-30.71, 28.9, -17.5) mm, rotated rx -180 ry 0 rz 90 deg; joints [74.476, -17.653, 86.792, 0, 20.861, 74.476]
  MoveC 9505 to (-31.07, 29.28, -17.5) mm, rotated rx 180 ry 0 rz 90 deg; joints [74.485, -17.661, 86.825, 0, 20.836, 74.485] to (-31.48, 29.6, -17.5) mm, rotated rx 180 ry 0 rz 90 deg; joints [74.492, -17.669, 86.859, 0, 20.81, 74.492]
  MoveC 9506 to (-48.16, 40.87, -17.5) mm, rotated rx 180 ry 0 rz 90 deg; joints [74.715, -17.986, 88.215, 0, 19.77, 74.715] to (-64.91, 52.03, -17.5) mm, rotated rx 180 ry 0 rz 90 deg; joints [74.939, -18.285, 89.553, 0, 18.732, 74.939]
  MoveC 9507 to (-66.96, 51.9, -17.5) mm, rotated rx -180 ry 0 rz 90 deg; joints [74.916, -18.314, 89.688, 0, 18.626, 74.916] to (-68.39, 50.43, -17.5) mm, rotated rx -180 ry 0 rz 90 deg; joints [74.852, -18.329, 89.757, 0, 18.572, 74.852]
  MoveL 9508 to (-68.4, 50.1, -17.5) mm, rotated rx 180 ry 0 rz 90 deg; joints [74.841, -18.328, 89.752, 0, 18.576, 74.841]
  MoveL 9509 to (-68.4, 28.48, -17.5) mm, rotated rx -180 ry 0 rz 90 deg; joints [74.107, -18.24, 89.349, 0, 18.891, 74.107]
  MoveL 9510 to (-60.85, 28.48, -17.5) mm, rotated rx -180 ry 0 rz 90 deg; joints [74.179, -18.127, 88.841, 0, 19.286, 74.179]
  MoveL 9511 to (-60.85, 28.48, -14.5) mm, rotated rx -180 ry 0 rz 90 deg; joints [74.179, -18.284, 88.944, 0, 19.34, 74.179]
  Establecer velocidad (1000.0 mm/s)
  MoveL 9512 to (-60.85, 28.48, 10) mm, rotated rx -180 ry 0 rz 90 deg; joints [74.179, -19.563, 89.769, 0, 19.795, 74.179]
  Establecer velocidad (66.7 mm/s)
  MoveL 9513 to (-41.46, -51.29, 10) mm, rotated rx 180 ry 0 rz 90 deg; joints [71.738, -18.843, 86.782, 0, 22.061, 71.738]
  MoveL 9514 to (-41.46, -51.29, -14.25) mm, rotated rx 180 ry 0 rz 90 deg; joints [71.738, -17.594, 85.967, 0, 21.627, 71.738]
  MoveL 9515 to (-40.05, -51.84, -14.66) mm, rotated rx -180 ry 0 rz 90 deg; joints [71.735, -17.546, 85.843, 0, 21.703, 71.735]
  MoveL 9516 to (-38.54, -52.03, -15.06) mm, rotated rx 180 ry 0 rz 90 deg; joints [71.745, -17.498, 85.721, 0, 21.777, 71.745]
  MoveL 9517 to (-37.03, -51.88, -15.47) mm, rotated rx 180 ry 0 rz 90 deg; joints [71.766, -17.452, 85.606, 0, 21.846, 71.766]
  MoveL 9518 to (-35.59, -51.4, -15.88) mm, rotated rx 180 ry 0 rz 90 deg; joints [71.797, -17.409, 85.503, 0, 21.906, 71.797]
  MoveL 9519 to (-34.28, -50.62, -16.28) mm, rotated rx 180 ry 0 rz 90 deg; joints [71.836, -17.37, 85.417, 0, 21.953, 71.836]
  MoveL 9520 to (-33.19, -49.57, -16.69) mm, rotated rx 180 ry 0 rz 90 deg; joints [71.882, -17.336, 85.351, 0, 21.985, 71.882]
  MoveL 9521 to (-32.35, -48.3, -17.09) mm, rotated rx -180 ry 0 rz 90 deg; joints [71.931, -17.308, 85.308, 0, 22, 71.931]
  MoveL 9522 to (-31.85, -46.87, -17.5) mm, rotated rx 180 ry 0 rz 90 deg; joints [71.983, -17.287, 85.292, 0, 21.995, 71.983]
  MoveL 9523 to (-28.91, -35.19, -17.5) mm, rotated rx 180 ry 0 rz 90 deg; joints [72.391, -17.301, 85.347, 0, 21.953, 72.391]
  MoveL 9524 to (-28.91, -27.8, -17.5) mm, rotated rx -180 ry 0 rz 90 deg; joints [72.632, -17.341, 85.509, 0, 21.832, 72.632]
  MoveC 9525 to (-29.51, -27.36, -17.5) mm, rotated rx -180 ry 0 rz 90 deg; joints [72.64, -17.353, 85.56, 0, 21.793, 72.64] to (-30.22, -27.16, -17.5) mm, rotated rx 180 ry 0 rz 90 deg; joints [72.639, -17.367, 85.614, 0, 21.753, 72.639]
  MoveC 9526 to (-48.42, -30.49, -17.5) mm, rotated rx -180 ry 0 rz 90 deg; joints [72.343, -17.653, 86.793, 0, 20.86, 72.343] to (-66.59, -33.96, -17.5) mm, rotated rx -180 ry 0 rz 90 deg; joints [72.036, -17.925, 87.95, 0, 19.975, 72.036]
  MoveC 9527 to (-67.87, -34.72, -17.5) mm, rotated rx -180 ry 0 rz 90 deg; joints [71.997, -17.941, 88.02, 0, 19.921, 71.997] to (-68.39, -36.11, -17.5) mm, rotated rx 180 ry 0 rz 90 deg; joints [71.946, -17.942, 88.024, 0, 19.918, 71.946]
  MoveL 9528 to (-68.4, -36.48, -17.5) mm, rotated rx 180 ry 0 rz 90 deg; joints [71.933, -17.94, 88.016, 0, 19.924, 71.933]
  MoveL 9529 to (-68.4, -65.86, -17.5) mm, rotated rx -180 ry 0 rz 90 deg; joints [70.967, -17.786, 87.353, 0, 20.433, 70.967]
  MoveL 9530 to (-68.39, -66.18, -17.5) mm, rotated rx -180 ry 0 rz 90 deg; joints [70.957, -17.784, 87.345, 0, 20.439, 70.957]
  MoveC 9531 to (-67.69, -67.79, -17.5) mm, rotated rx -180 ry 0 rz 90 deg; joints [70.912, -17.764, 87.261, 0, 20.503, 70.912] to (-66.06, -68.42, -17.5) mm, rotated rx -180 ry 0 rz 90 deg; joints [70.91, -17.735, 87.136, 0, 20.599, 70.91]
  MoveC 9532 to (-52.45, -68.04, -17.5) mm, rotated rx 180 ry 0 rz 90 deg; joints [71.075, -17.515, 86.221, 0, 21.294, 71.075] to (-38.84, -67.57, -17.5) mm, rotated rx -180 ry 0 rz 90 deg; joints [71.24, -17.288, 85.299, 0, 21.989, 71.24]
  MoveC 9533 to (-38.53, -67.54, -17.5) mm, rotated rx 180 ry 0 rz 90 deg; joints [71.244, -17.283, 85.278, 0, 22.005, 71.244] to (-38.23, -67.46, -17.5) mm, rotated rx 180 ry 0 rz 90 deg; joints [71.25, -17.279, 85.259, 0, 22.019, 71.25]
  MoveC 9534 to (-37.19, -66.79, -17.5) mm, rotated rx -180 ry 0 rz 90 deg; joints [71.283, -17.265, 85.203, 0, 22.061, 71.283] to (-36.6, -65.71, -17.5) mm, rotated rx 180 ry 0 rz 90 deg; joints [71.324, -17.261, 85.188, 0, 22.073, 71.324]
  MoveL 9535 to (-31.85, -46.87, -17.5) mm, rotated rx 180 ry 0 rz 90 deg; joints [71.983, -17.287, 85.292, 0, 21.995, 71.983]
  MoveL 9536 to (-39.17, -45.02, -17.5) mm, rotated rx 180 ry 0 rz 90 deg; joints [71.966, -17.422, 85.839, 0, 21.583, 71.966]
  MoveL 9537 to (-39.17, -45.02, -14.5) mm, rotated rx 180 ry 0 rz 90 deg; joints [71.966, -17.577, 85.942, 0, 21.635, 71.966]
  Establecer velocidad (1000.0 mm/s)
  MoveL 9538 to (-39.17, -45.02, 10) mm, rotated rx 180 ry 0 rz 90 deg; joints [71.966, -18.839, 86.766, 0, 22.073, 71.966]
  Establecer velocidad (66.7 mm/s)
  MoveL 9539 to (-41.61, -51.25, 10) mm, rotated rx 180 ry 0 rz 90 deg; joints [71.738, -18.846, 86.793, 0, 22.053, 71.738]
  MoveL 9540 to (-41.61, -51.25, -14.5) mm, rotated rx 180 ry 0 rz 90 deg; joints [71.738, -17.583, 85.969, 0, 21.614, 71.738]
  MoveL 9541 to (-40.19, -51.8, -14.91) mm, rotated rx -180 ry 0 rz 90 deg; joints [71.735, -17.535, 85.845, 0, 21.69, 71.735]
  MoveL 9542 to (-38.68, -51.99, -15.31) mm, rotated rx 180 ry 0 rz 90 deg; joints [71.745, -17.488, 85.723, 0, 21.765, 71.745]
  MoveL 9543 to (-37.17, -51.84, -15.72) mm, rotated rx 180 ry 0 rz 90 deg; joints [71.766, -17.442, 85.608, 0, 21.834, 71.766]
  MoveL 9544 to (-35.73, -51.37, -16.12) mm, rotated rx 180 ry 0 rz 90 deg; joints [71.796, -17.399, 85.506, 0, 21.893, 71.796]
  MoveL 9545 to (-34.43, -50.58, -16.53) mm, rotated rx 180 ry 0 rz 90 deg; joints [71.836, -17.36, 85.419, 0, 21.941, 71.836]
  MoveL 9546 to (-33.33, -49.53, -16.94) mm, rotated rx -180 ry 0 rz 90 deg; joints [71.881, -17.326, 85.354, 0, 21.973, 71.881]
  MoveL 9547 to (-32.5, -48.26, -17.34) mm, rotated rx 180 ry 0 rz 90 deg; joints [71.931, -17.298, 85.31, 0, 21.988, 71.931]
  MoveL 9548 to (-31.99, -46.83, -17.75) mm, rotated rx 180 ry 0 rz 90 deg; joints [71.983, -17.276, 85.294, 0, 21.983, 71.983]
  MoveL 9549 to (-31.76, -45.92, -17.75) mm, rotated rx -180 ry 0 rz 90 deg; joints [72.014, -17.278, 85.298, 0, 21.979, 72.014]
  MoveL 9550 to (-31.76, -27.61, -17.75) mm, rotated rx -180 ry 0 rz 90 deg; joints [72.608, -17.378, 85.703, 0, 21.675, 72.608]
  MoveC 9551 to (-49.11, -30.78, -17.75) mm, rotated rx -180 ry 0 rz 90 deg; joints [72.326, -17.65, 86.826, 0, 20.824, 72.326] to (-66.44, -34.08, -17.75) mm, rotated rx -180 ry 0 rz 90 deg; joints [72.034, -17.909, 87.929, 0, 19.98, 72.034]
  MoveC 9552 to (-67.72, -34.84, -17.75) mm, rotated rx 180 ry 0 rz 90 deg; joints [71.995, -17.925, 87.998, 0, 19.927, 71.995] to (-68.23, -36.25, -17.75) mm, rotated rx -180 ry 0 rz 90 deg; joints [71.943, -17.926, 88.002, 0, 19.924, 71.943]
  MoveL 9553 to (-68.23, -37.43, -17.75) mm, rotated rx 180 ry 0 rz 90 deg; joints [71.904, -17.92, 87.976, 0, 19.944, 71.904]
  MoveL 9554 to (-68.23, -64.91, -17.75) mm, rotated rx 180 ry 0 rz 90 deg; joints [71, -17.775, 87.356, 0, 20.42, 71]
  MoveL 9555 to (-68.23, -66.01, -17.75) mm, rotated rx -180 ry 0 rz 90 deg; joints [70.964, -17.769, 87.33, 0, 20.44, 70.964]
  MoveC 9556 to (-67.54, -67.63, -17.75) mm, rotated rx -180 ry 0 rz 90 deg; joints [70.919, -17.75, 87.246, 0, 20.504, 70.919] to (-65.9, -68.28, -17.75) mm, rotated rx 180 ry 0 rz 90 deg; joints [70.917, -17.72, 87.12, 0, 20.6, 70.917]
  MoveC 9557 to (-52.61, -67.89, -17.75) mm, rotated rx 180 ry 0 rz 90 deg; joints [71.078, -17.506, 86.228, 0, 21.279, 71.078] to (-39.33, -67.42, -17.75) mm, rotated rx -180 ry 0 rz 90 deg; joints [71.239, -17.285, 85.327, 0, 21.957, 71.239]
  MoveL 9558 to (-38.69, -67.35, -17.75) mm, rotated rx 180 ry 0 rz 90 deg; joints [71.249, -17.274, 85.285, 0, 21.989, 71.249]
  MoveC 9559 to (-37.49, -66.83, -17.75) mm, rotated rx 180 ry 0 rz 90 deg; joints [71.279, -17.257, 85.214, 0, 22.042, 71.279] to (-36.78, -65.73, -17.75) mm, rotated rx -180 ry 0 rz 90 deg; joints [71.322, -17.251, 85.191, 0, 22.06, 71.322]
  MoveL 9560 to (-36.55, -64.91, -17.75) mm, rotated rx 180 ry 0 rz 90 deg; joints [71.35, -17.252, 85.195, 0, 22.057, 71.35]
  MoveL 9561 to (-34.64, -57.33, -17.75) mm, rotated rx -180 ry 0 rz 90 deg; joints [71.615, -17.263, 85.238, 0, 22.025, 71.615]
  MoveL 9562 to (-34.4, -56.39, -17.75) mm, rotated rx -180 ry 0 rz 90 deg; joints [71.648, -17.264, 85.243, 0, 22.021, 71.648]
  MoveL 9563 to (-34.17, -55.44, -17.75) mm, rotated rx 180 ry 0 rz 90 deg; joints [71.682, -17.265, 85.249, 0, 22.017, 71.682]
  MoveL 9564 to (-31.99, -46.83, -17.75) mm, rotated rx 180 ry 0 rz 90 deg; joints [71.983, -17.276, 85.294, 0, 21.983, 71.983]
  MoveL 9565 to (-39.31, -44.98, -17.75) mm, rotated rx 180 ry 0 rz 90 deg; joints [71.965, -17.412, 85.841, 0, 21.571, 71.965]
  MoveL 9566 to (-39.31, -44.98, -14.75) mm, rotated rx 180 ry 0 rz 90 deg; joints [71.965, -17.567, 85.944, 0, 21.623, 71.965]
  Establecer velocidad (1000.0 mm/s)
  MoveL 9567 to (-39.31, -44.98, 10) mm, rotated rx -180 ry 0 rz 90 deg; joints [71.965, -18.842, 86.776, 0, 22.065, 71.965]
  Establecer velocidad (66.7 mm/s)
  MoveL 9568 to (-59.99, 35.04, 10) mm, rotated rx -180 ry 0 rz 90 deg; joints [74.409, -19.579, 89.836, 0, 19.743, 74.409]
  MoveL 9569 to (-59.99, 35.04, -14.5) mm, rotated rx 180 ry 0 rz 90 deg; joints [74.409, -18.299, 89.011, 0, 19.288, 74.409]
  MoveL 9570 to (-61.5, 35.23, -14.91) mm, rotated rx 180 ry 0 rz 90 deg; joints [74.401, -18.301, 89.103, 0, 19.199, 74.401]
  MoveL 9571 to (-63.01, 35.04, -15.31) mm, rotated rx 180 ry 0 rz 90 deg; joints [74.38, -18.302, 89.187, 0, 19.115, 74.38]
  MoveL 9572 to (-64.44, 34.53, -15.72) mm, rotated rx -180 ry 0 rz 90 deg; joints [74.349, -18.3, 89.259, 0, 19.041, 74.349]
  MoveL 9573 to (-65.72, 33.72, -16.12) mm, rotated rx 180 ry 0 rz 90 deg; joints [74.31, -18.294, 89.316, 0, 18.978, 74.31]
  MoveL 9574 to (-66.79, 32.64, -16.53) mm, rotated rx -180 ry 0 rz 90 deg; joints [74.263, -18.284, 89.354, 0, 18.931, 74.263]
  MoveL 9575 to (-67.6, 31.35, -16.94) mm, rotated rx 180 ry 0 rz 90 deg; joints [74.211, -18.27, 89.369, 0, 18.9, 74.211]
  MoveL 9576 to (-68.09, 29.91, -17.34) mm, rotated rx 180 ry 0 rz 90 deg; joints [74.158, -18.25, 89.361, 0, 18.888, 74.158]
  MoveL 9577 to (-68.23, 28.4, -17.75) mm, rotated rx -180 ry 0 rz 90 deg; joints [74.106, -18.224, 89.328, 0, 18.896, 74.106]
  MoveL 9578 to (-68.23, 7.11, -17.75) mm, rotated rx 180 ry 0 rz 90 deg; joints [73.388, -18.132, 88.911, 0, 19.22, 73.388]
  MoveL 9579 to (-68.23, 6.63, -17.75) mm, rotated rx -180 ry 0 rz 90 deg; joints [73.372, -18.13, 88.902, 0, 19.228, 73.372]
  MoveC 9580 to (-67.28, 4.95, -17.75) mm, rotated rx -180 ry 0 rz 90 deg; joints [73.325, -18.108, 88.804, 0, 19.304, 73.325] to (-65.39, 4.55, -17.75) mm, rotated rx -180 ry 0 rz 90 deg; joints [73.331, -18.077, 88.669, 0, 19.409, 73.331]
  MoveC 9581 to (-48.56, 8.79, -17.75) mm, rotated rx -180 ry 0 rz 90 deg; joints [73.639, -17.836, 87.614, 0, 20.222, 73.639] to (-31.76, 13.16, -17.75) mm, rotated rx 180 ry 0 rz 90 deg; joints [73.945, -17.584, 86.549, 0, 21.034, 73.945]
  MoveL 9582 to (-31.76, 29.6, -17.75) mm, rotated rx 180 ry 0 rz 90 deg; joints [74.49, -17.661, 86.87, 0, 20.79, 74.49]
  MoveC 9583 to (-46.88, 39.84, -17.75) mm, rotated rx -180 ry 0 rz 90 deg; joints [74.692, -17.948, 88.1, 0, 19.848, 74.692] to (-62.07, 49.98, -17.75) mm, rotated rx -180 ry 0 rz 90 deg; joints [74.895, -18.221, 89.316, 0, 18.905, 74.895]
  MoveL 9584 to (-63.02, 50.61, -17.75) mm, rotated rx 180 ry 0 rz 90 deg; joints [74.908, -18.238, 89.391, 0, 18.847, 74.908]
  MoveL 9585 to (-64.57, 51.65, -17.75) mm, rotated rx 180 ry 0 rz 90 deg; joints [74.929, -18.265, 89.514, 0, 18.751, 74.929]
  MoveL 9586 to (-64.91, 51.85, -17.75) mm, rotated rx 180 ry 0 rz 90 deg; joints [74.933, -18.271, 89.541, 0, 18.73, 74.933]
  MoveC 9587 to (-66.88, 51.62, -17.75) mm, rotated rx 180 ry 0 rz 90 deg; joints [74.907, -18.299, 89.669, 0, 18.629, 74.907] to (-68.23, 50.17, -17.75) mm, rotated rx -180 ry 0 rz 90 deg; joints [74.845, -18.313, 89.733, 0, 18.579, 74.845]
  MoveL 9588 to (-68.23, 49.88, -17.75) mm, rotated rx 180 ry 0 rz 90 deg; joints [74.835, -18.312, 89.728, 0, 18.583, 74.835]
  MoveL 9589 to (-68.23, 28.4, -17.75) mm, rotated rx -180 ry 0 rz 90 deg; joints [74.106, -18.224, 89.328, 0, 18.896, 74.106]
  MoveL 9590 to (-60.69, 28.4, -17.75) mm, rotated rx 180 ry 0 rz 90 deg; joints [74.178, -18.111, 88.82, 0, 19.291, 74.178]
  MoveL 9591 to (-60.69, 28.4, -14.75) mm, rotated rx -180 ry 0 rz 90 deg; joints [74.178, -18.268, 88.923, 0, 19.345, 74.178]
  Establecer velocidad (1000.0 mm/s)
  MoveL 9592 to (-60.69, 28.4, 10) mm, rotated rx 180 ry 0 rz 90 deg; joints [74.178, -19.561, 89.756, 0, 19.804, 74.178]
  Establecer velocidad (66.7 mm/s)
  MoveL 9593 to (-59.83, 35.04, 10) mm, rotated rx 180 ry 0 rz 90 deg; joints [74.41, -19.576, 89.825, 0, 19.752, 74.41]
  MoveL 9594 to (-59.83, 35.04, -14.75) mm, rotated rx -180 ry 0 rz 90 deg; joints [74.41, -18.284, 88.992, 0, 19.292, 74.41]
  MoveL 9595 to (-61.34, 35.23, -15.16) mm, rotated rx -180 ry 0 rz 90 deg; joints [74.402, -18.286, 89.083, 0, 19.203, 74.402]
  MoveL 9596 to (-62.84, 35.04, -15.56) mm, rotated rx 180 ry 0 rz 90 deg; joints [74.382, -18.286, 89.167, 0, 19.119, 74.382]
  MoveL 9597 to (-64.27, 34.53, -15.97) mm, rotated rx 180 ry 0 rz 90 deg; joints [74.351, -18.284, 89.24, 0, 19.045, 74.351]
  MoveL 9598 to (-65.56, 33.72, -16.38) mm, rotated rx 180 ry 0 rz 90 deg; joints [74.311, -18.279, 89.297, 0, 18.982, 74.311]
  MoveL 9599 to (-66.63, 32.64, -16.78) mm, rotated rx 180 ry 0 rz 90 deg; joints [74.264, -18.269, 89.334, 0, 18.935, 74.264]
  MoveL 9600 to (-67.43, 31.35, -17.19) mm, rotated rx 180 ry 0 rz 90 deg; joints [74.213, -18.254, 89.35, 0, 18.904, 74.213]
  MoveL 9601 to (-67.93, 29.91, -17.59) mm, rotated rx -180 ry 0 rz 90 deg; joints [74.16, -18.234, 89.342, 0, 18.892, 74.16]
  MoveL 9602 to (-68.07, 28.4, -18) mm, rotated rx 180 ry 0 rz 90 deg; joints [74.107, -18.209, 89.308, 0, 18.9, 74.107]
  MoveL 9603 to (-68.07, 7.11, -18) mm, rotated rx -180 ry 0 rz 90 deg; joints [73.389, -18.116, 88.892, 0, 19.224, 73.389]
  MoveL 9604 to (-68.05, 6.63, -18) mm, rotated rx 180 ry 0 rz 90 deg; joints [73.374, -18.114, 88.881, 0, 19.233, 73.374]
  MoveC 9605 to (-67.03, 5.06, -18) mm, rotated rx 180 ry 0 rz 90 deg; joints [73.331, -18.091, 88.781, 0, 19.31, 73.331] to (-65.18, 4.74, -18) mm, rotated rx -180 ry 0 rz 90 deg; joints [73.339, -18.062, 88.65, 0, 19.412, 73.339]
  MoveC 9606 to (-49.89, 8.6, -18) mm, rotated rx -180 ry 0 rz 90 deg; joints [73.619, -17.843, 87.692, 0, 20.151, 73.619] to (-34.62, 12.58, -18) mm, rotated rx 180 ry 0 rz 90 deg; joints [73.899, -17.615, 86.726, 0, 20.889, 73.899]
  MoveL 9607 to (-34.62, 31.36, -18) mm, rotated rx -180 ry 0 rz 90 deg; joints [74.522, -17.702, 87.092, 0, 20.61, 74.522]
  MoveC 9608 to (-49.66, 41.54, -18) mm, rotated rx -180 ry 0 rz 90 deg; joints [74.724, -17.986, 88.313, 0, 19.673, 74.724] to (-64.78, 51.61, -18) mm, rotated rx 180 ry 0 rz 90 deg; joints [74.926, -18.255, 89.519, 0, 18.736, 74.926]
  MoveC 9609 to (-66.36, 51.53, -18) mm, rotated rx -180 ry 0 rz 90 deg; joints [74.908, -18.278, 89.624, 0, 18.654, 74.908] to (-67.68, 50.64, -18) mm, rotated rx 180 ry 0 rz 90 deg; joints [74.866, -18.293, 89.696, 0, 18.597, 74.866]
  MoveC 9610 to (-67.97, 50.15, -18) mm, rotated rx -180 ry 0 rz 90 deg; joints [74.847, -18.296, 89.707, 0, 18.589, 74.847] to (-68.07, 49.6, -18) mm, rotated rx 180 ry 0 rz 90 deg; joints [74.827, -18.295, 89.703, 0, 18.591, 74.827]
  MoveL 9611 to (-68.07, 28.4, -18) mm, rotated rx 180 ry 0 rz 90 deg; joints [74.107, -18.209, 89.308, 0, 18.9, 74.107]
  MoveL 9612 to (-60.52, 28.4, -18) mm, rotated rx -180 ry 0 rz 90 deg; joints [74.18, -18.096, 88.8, 0, 19.295, 74.18]
  MoveL 9613 to (-60.52, 28.4, -15) mm, rotated rx 180 ry 0 rz 90 deg; joints [74.18, -18.253, 88.904, 0, 19.349, 74.18]
  Establecer velocidad (1000.0 mm/s)
  MoveL 9614 to (-60.52, 28.4, 10) mm, rotated rx -180 ry 0 rz 90 deg; joints [74.18, -19.558, 89.745, 0, 19.813, 74.18]
  Establecer velocidad (66.7 mm/s)
  MoveL 9615 to (-42.86, -53.87, 10) mm, rotated rx -180 ry 0 rz 90 deg; joints [71.639, -18.852, 86.819, 0, 22.033, 71.639]
  MoveL 9616 to (-42.86, -53.87, -14.75) mm, rotated rx 180 ry 0 rz 90 deg; joints [71.639, -17.577, 85.987, 0, 21.59, 71.639]
  MoveL 9617 to (-41.35, -54.05, -15.16) mm, rotated rx -180 ry 0 rz 90 deg; joints [71.649, -17.53, 85.865, 0, 21.664, 71.649]
  MoveL 9618 to (-39.84, -53.87, -15.56) mm, rotated rx 180 ry 0 rz 90 deg; joints [71.671, -17.484, 85.752, 0, 21.732, 71.671]
  MoveL 9619 to (-38.41, -53.36, -15.97) mm, rotated rx -180 ry 0 rz 90 deg; joints [71.703, -17.442, 85.651, 0, 21.791, 71.703]
  MoveL 9620 to (-37.13, -52.54, -16.38) mm, rotated rx 180 ry 0 rz 90 deg; joints [71.743, -17.403, 85.567, 0, 21.836, 71.743]
  MoveL 9621 to (-36.06, -51.46, -16.78) mm, rotated rx 180 ry 0 rz 90 deg; joints [71.79, -17.37, 85.504, 0, 21.867, 71.79]
  MoveL 9622 to (-35.26, -50.18, -17.19) mm, rotated rx 180 ry 0 rz 90 deg; joints [71.84, -17.343, 85.463, 0, 21.879, 71.84]
  MoveL 9623 to (-34.76, -48.74, -17.59) mm, rotated rx -180 ry 0 rz 90 deg; joints [71.892, -17.321, 85.447, 0, 21.874, 71.892]
  MoveL 9624 to (-34.62, -47.23, -18) mm, rotated rx 180 ry 0 rz 90 deg; joints [71.942, -17.306, 85.458, 0, 21.849, 71.942]
  MoveL 9625 to (-34.62, -28.3, -18) mm, rotated rx 180 ry 0 rz 90 deg; joints [72.557, -17.41, 85.876, 0, 21.533, 72.557]
  MoveC 9626 to (-50.46, -31.2, -18) mm, rotated rx 180 ry 0 rz 90 deg; joints [72.298, -17.657, 86.901, 0, 20.756, 72.298] to (-66.29, -34.21, -18) mm, rotated rx 180 ry 0 rz 90 deg; joints [72.031, -17.893, 87.907, 0, 19.986, 72.031]
  MoveC 9627 to (-67.56, -34.96, -18) mm, rotated rx -180 ry 0 rz 90 deg; joints [71.993, -17.909, 87.976, 0, 19.932, 71.993] to (-68.06, -36.34, -18) mm, rotated rx 180 ry 0 rz 90 deg; joints [71.941, -17.91, 87.98, 0, 19.93, 71.941]
  MoveL 9628 to (-68.07, -37.43, -18) mm, rotated rx -180 ry 0 rz 90 deg; joints [71.905, -17.904, 87.956, 0, 19.948, 71.905]
  MoveL 9629 to (-68.07, -64.91, -18) mm, rotated rx 180 ry 0 rz 90 deg; joints [71.002, -17.76, 87.336, 0, 20.424, 71.002]
  MoveL 9630 to (-68.07, -65.86, -18) mm, rotated rx 180 ry 0 rz 90 deg; joints [70.971, -17.755, 87.314, 0, 20.441, 70.971]
  MoveC 9631 to (-67.43, -67.45, -18) mm, rotated rx 180 ry 0 rz 90 deg; joints [70.926, -17.736, 87.234, 0, 20.502, 70.926] to (-65.86, -68.12, -18) mm, rotated rx -180 ry 0 rz 90 deg; joints [70.922, -17.707, 87.112, 0, 20.595, 70.922]
  MoveC 9632 to (-52.59, -67.74, -18) mm, rotated rx 180 ry 0 rz 90 deg; joints [71.083, -17.494, 86.221, 0, 21.273, 71.083] to (-39.33, -67.26, -18) mm, rotated rx 180 ry 0 rz 90 deg; joints [71.245, -17.273, 85.323, 0, 21.95, 71.245]
  MoveL 9633 to (-38.38, -67.13, -18) mm, rotated rx 180 ry 0 rz 90 deg; joints [71.259, -17.257, 85.26, 0, 21.997, 71.259]
  MoveC 9634 to (-37.56, -66.63, -18) mm, rotated rx -180 ry 0 rz 90 deg; joints [71.284, -17.246, 85.215, 0, 22.031, 71.284] to (-36.98, -65.86, -18) mm, rotated rx 180 ry 0 rz 90 deg; joints [71.315, -17.241, 85.193, 0, 22.047, 71.315]
  MoveL 9635 to (-36.7, -64.91, -18) mm, rotated rx -180 ry 0 rz 90 deg; joints [71.349, -17.241, 85.196, 0, 22.045, 71.349]
  MoveL 9636 to (-34.62, -56.65, -18) mm, rotated rx 180 ry 0 rz 90 deg; joints [71.638, -17.253, 85.244, 0, 22.01, 71.638]
  MoveL 9637 to (-34.62, -47.23, -18) mm, rotated rx 180 ry 0 rz 90 deg; joints [71.942, -17.306, 85.458, 0, 21.849, 71.942]
  MoveL 9638 to (-42.17, -47.23, -18) mm, rotated rx 180 ry 0 rz 90 deg; joints [71.862, -17.434, 85.978, 0, 21.456, 71.862]
  MoveL 9639 to (-42.17, -47.23, -15) mm, rotated rx 180 ry 0 rz 90 deg; joints [71.862, -17.589, 86.081, 0, 21.508, 71.862]
  Establecer velocidad (1000.0 mm/s)
  MoveL 9640 to (-42.17, -47.23, 10) mm, rotated rx -180 ry 0 rz 90 deg; joints [71.862, -18.878, 86.922, 0, 21.956, 71.862]
  Establecer velocidad (66.7 mm/s)
  MoveL 9641 to (-45.72, -53.87, 10) mm, rotated rx -180 ry 0 rz 90 deg; joints [71.608, -18.902, 87.015, 0, 21.886, 71.608]
  MoveL 9642 to (-45.72, -53.87, -15) mm, rotated rx -180 ry 0 rz 90 deg; joints [71.608, -17.612, 86.174, 0, 21.438, 71.608]
  MoveL 9643 to (-44.21, -54.05, -15.41) mm, rotated rx -180 ry 0 rz 90 deg; joints [71.619, -17.565, 86.053, 0, 21.512, 71.619]
  MoveL 9644 to (-42.7, -53.87, -15.81) mm, rotated rx 180 ry 0 rz 90 deg; joints [71.641, -17.52, 85.94, 0, 21.58, 71.641]
  MoveL 9645 to (-41.27, -53.36, -16.22) mm, rotated rx 180 ry 0 rz 90 deg; joints [71.673, -17.477, 85.839, 0, 21.638, 71.673]
  MoveL 9646 to (-39.99, -52.54, -16.62) mm, rotated rx 180 ry 0 rz 90 deg; joints [71.713, -17.439, 85.755, 0, 21.684, 71.713]
  MoveL 9647 to (-38.92, -51.46, -17.03) mm, rotated rx 180 ry 0 rz 90 deg; joints [71.759, -17.406, 85.692, 0, 21.714, 71.759]
  MoveL 9648 to (-38.12, -50.18, -17.44) mm, rotated rx 180 ry 0 rz 90 deg; joints [71.81, -17.379, 85.652, 0, 21.727, 71.81]
  MoveL 9649 to (-37.62, -48.74, -17.84) mm, rotated rx -180 ry 0 rz 90 deg; joints [71.861, -17.357, 85.636, 0, 21.721, 71.861]
  MoveL 9650 to (-37.48, -47.23, -18.25) mm, rotated rx 180 ry 0 rz 90 deg; joints [71.912, -17.342, 85.647, 0, 21.696, 71.912]
  MoveL 9651 to (-37.48, -28.99, -18.25) mm, rotated rx 180 ry 0 rz 90 deg; joints [72.505, -17.441, 86.05, 0, 21.391, 72.505]
  MoveL 9652 to (-41.22, -29.66, -18.25) mm, rotated rx 180 ry 0 rz 90 deg; joints [72.444, -17.5, 86.293, 0, 21.207, 72.444]
  MoveL 9653 to (-61.12, -33.36, -18.25) mm, rotated rx 180 ry 0 rz 90 deg; joints [72.114, -17.803, 87.569, 0, 20.235, 72.114]
  MoveL 9654 to (-66.15, -34.33, -18.25) mm, rotated rx 180 ry 0 rz 90 deg; joints [72.029, -17.877, 87.887, 0, 19.99, 72.029]
  MoveC 9655 to (-67.4, -35.07, -18.25) mm, rotated rx -180 ry 0 rz 90 deg; joints [71.991, -17.893, 87.955, 0, 19.938, 71.991] to (-67.9, -36.43, -18.25) mm, rotated rx -180 ry 0 rz 90 deg; joints [71.94, -17.894, 87.958, 0, 19.935, 71.94]
  MoveL 9656 to (-67.91, -37.43, -18.25) mm, rotated rx 180 ry 0 rz 90 deg; joints [71.907, -17.889, 87.937, 0, 19.952, 71.907]
  MoveL 9657 to (-67.91, -64.91, -18.25) mm, rotated rx -180 ry 0 rz 90 deg; joints [71.004, -17.744, 87.316, 0, 20.428, 71.004]
  MoveL 9658 to (-67.9, -65.8, -18.25) mm, rotated rx 180 ry 0 rz 90 deg; joints [70.975, -17.739, 87.295, 0, 20.444, 70.975]
  MoveC 9659 to (-67.24, -67.35, -18.25) mm, rotated rx -180 ry 0 rz 90 deg; joints [70.932, -17.72, 87.215, 0, 20.506, 70.932] to (-65.67, -67.97, -18.25) mm, rotated rx -180 ry 0 rz 90 deg; joints [70.929, -17.692, 87.094, 0, 20.598, 70.929]
  MoveC 9660 to (-52.39, -67.58, -18.25) mm, rotated rx -180 ry 0 rz 90 deg; joints [71.09, -17.478, 86.203, 0, 21.276, 71.09] to (-39.12, -67.09, -18.25) mm, rotated rx -180 ry 0 rz 90 deg; joints [71.253, -17.258, 85.304, 0, 21.954, 71.253]
  MoveC 9661 to (-38.22, -66.86, -18.25) mm, rotated rx -180 ry 0 rz 90 deg; joints [71.27, -17.243, 85.247, 0, 21.996, 71.27] to (-37.48, -66.3, -18.25) mm, rotated rx 180 ry 0 rz 90 deg; joints [71.296, -17.234, 85.209, 0, 22.025, 71.296]
  MoveL 9662 to (-37.48, -47.23, -18.25) mm, rotated rx 180 ry 0 rz 90 deg; joints [71.912, -17.342, 85.647, 0, 21.696, 71.912]
  MoveL 9663 to (-45.03, -47.23, -18.25) mm, rotated rx -180 ry 0 rz 90 deg; joints [71.832, -17.469, 86.166, 0, 21.304, 71.832]
  MoveL 9664 to (-45.03, -47.23, -15.25) mm, rotated rx 180 ry 0 rz 90 deg; joints [71.832, -17.624, 86.269, 0, 21.356, 71.832]
  Establecer velocidad (1000.0 mm/s)
  MoveL 9665 to (-45.03, -47.23, 10) mm, rotated rx -180 ry 0 rz 90 deg; joints [71.832, -18.927, 87.118, 0, 21.809, 71.832]
  Establecer velocidad (66.7 mm/s)
  MoveL 9666 to (-59.67, 35.1, 10) mm, rotated rx -180 ry 0 rz 90 deg; joints [74.413, -19.574, 89.815, 0, 19.759, 74.413]
  MoveL 9667 to (-59.67, 35.1, -15) mm, rotated rx 180 ry 0 rz 90 deg; joints [74.413, -18.268, 88.973, 0, 19.295, 74.413]
  MoveL 9668 to (-61.17, 35.28, -15.41) mm, rotated rx -180 ry 0 rz 90 deg; joints [74.406, -18.271, 89.064, 0, 19.206, 74.406]
  MoveL 9669 to (-62.68, 35.1, -15.81) mm, rotated rx 180 ry 0 rz 90 deg; joints [74.385, -18.271, 89.148, 0, 19.123, 74.385]
  MoveL 9670 to (-64.11, 34.58, -16.22) mm, rotated rx -180 ry 0 rz 90 deg; joints [74.354, -18.269, 89.221, 0, 19.048, 74.354]
  MoveL 9671 to (-65.39, 33.77, -16.62) mm, rotated rx -180 ry 0 rz 90 deg; joints [74.314, -18.263, 89.278, 0, 18.985, 74.314]
  MoveL 9672 to (-66.46, 32.69, -17.03) mm, rotated rx -180 ry 0 rz 90 deg; joints [74.268, -18.254, 89.316, 0, 18.938, 74.268]
  MoveL 9673 to (-67.27, 31.4, -17.44) mm, rotated rx 180 ry 0 rz 90 deg; joints [74.216, -18.239, 89.331, 0, 18.908, 74.216]
  MoveL 9674 to (-67.77, 29.96, -17.84) mm, rotated rx 180 ry 0 rz 90 deg; joints [74.163, -18.219, 89.323, 0, 18.896, 74.163]
  MoveL 9675 to (-67.91, 28.46, -18.25) mm, rotated rx 180 ry 0 rz 90 deg; joints [74.111, -18.193, 89.29, 0, 18.903, 74.111]
  MoveL 9676 to (-67.91, 6.98, -18.25) mm, rotated rx -180 ry 0 rz 90 deg; joints [73.387, -18.1, 88.87, 0, 19.231, 73.387]
  MoveC 9677 to (-67.74, 6.22, -18.25) mm, rotated rx -180 ry 0 rz 90 deg; joints [73.363, -18.094, 88.843, 0, 19.251, 73.363] to (-67.28, 5.59, -18.25) mm, rotated rx 180 ry 0 rz 90 deg; joints [73.346, -18.085, 88.8, 0, 19.285, 73.346]
  MoveC 9678 to (-66.29, 4.94, -18.25) mm, rotated rx 180 ry 0 rz 90 deg; joints [73.335, -18.067, 88.72, 0, 19.346, 73.335] to (-65.11, 4.91, -18.25) mm, rotated rx 180 ry 0 rz 90 deg; joints [73.345, -18.049, 88.64, 0, 19.409, 73.345]
  MoveC 9679 to (-51.28, 8.41, -18.25) mm, rotated rx 180 ry 0 rz 90 deg; joints [73.599, -17.851, 87.775, 0, 20.076, 73.599] to (-37.48, 12, -18.25) mm, rotated rx -180 ry 0 rz 90 deg; joints [73.852, -17.647, 86.903, 0, 20.744, 73.852]
  MoveL 9680 to (-37.48, 33.12, -18.25) mm, rotated rx 180 ry 0 rz 90 deg; joints [74.554, -17.744, 87.313, 0, 20.43, 74.554]
  MoveC 9681 to (-51.03, 42.29, -18.25) mm, rotated rx -180 ry 0 rz 90 deg; joints [74.736, -17.997, 88.411, 0, 19.586, 74.736] to (-64.65, 51.36, -18.25) mm, rotated rx -180 ry 0 rz 90 deg; joints [74.918, -18.239, 89.497, 0, 18.742, 74.918]
  MoveC 9682 to (-66.48, 51.18, -18.25) mm, rotated rx -180 ry 0 rz 90 deg; joints [74.895, -18.265, 89.617, 0, 18.648, 74.895] to (-67.83, 49.92, -18.25) mm, rotated rx 180 ry 0 rz 90 deg; joints [74.84, -18.28, 89.685, 0, 18.595, 74.84]
  MoveL 9683 to (-67.89, 49.75, -18.25) mm, rotated rx 180 ry 0 rz 90 deg; joints [74.834, -18.28, 89.686, 0, 18.594, 74.834]
  MoveL 9684 to (-67.91, 48.8, -18.25) mm, rotated rx -180 ry 0 rz 90 deg; joints [74.801, -18.276, 89.669, 0, 18.607, 74.801]
  MoveL 9685 to (-67.91, 28.46, -18.25) mm, rotated rx 180 ry 0 rz 90 deg; joints [74.111, -18.193, 89.29, 0, 18.903, 74.111]
  MoveL 9686 to (-60.36, 28.46, -18.25) mm, rotated rx -180 ry 0 rz 90 deg; joints [74.183, -18.081, 88.782, 0, 19.299, 74.183]
  MoveL 9687 to (-60.36, 28.46, -15.25) mm, rotated rx -180 ry 0 rz 90 deg; joints [74.183, -18.237, 88.885, 0, 19.352, 74.183]
  Establecer velocidad (1000.0 mm/s)
  MoveL 9688 to (-60.36, 28.46, 10) mm, rotated rx -180 ry 0 rz 90 deg; joints [74.183, -19.556, 89.735, 0, 19.821, 74.183]
  Establecer velocidad (66.7 mm/s)
  MoveL 9689 to (-59.5, 35.1, 10) mm, rotated rx -180 ry 0 rz 90 deg; joints [74.415, -19.571, 89.803, 0, 19.768, 74.415]
  MoveL 9690 to (-59.5, 35.1, -15.25) mm, rotated rx 180 ry 0 rz 90 deg; joints [74.415, -18.253, 88.953, 0, 19.299, 74.415]
  MoveL 9691 to (-61.01, 35.28, -15.66) mm, rotated rx -180 ry 0 rz 90 deg; joints [74.407, -18.255, 89.045, 0, 19.21, 74.407]
  MoveL 9692 to (-62.52, 35.1, -16.06) mm, rotated rx 180 ry 0 rz 90 deg; joints [74.387, -18.256, 89.129, 0, 19.127, 74.387]
  MoveL 9693 to (-63.95, 34.58, -16.47) mm, rotated rx 180 ry 0 rz 90 deg; joints [74.356, -18.253, 89.201, 0, 19.052, 74.356]
  MoveL 9694 to (-65.23, 33.77, -16.88) mm, rotated rx 180 ry 0 rz 90 deg; joints [74.316, -18.248, 89.258, 0, 18.99, 74.316]
  MoveL 9695 to (-66.3, 32.69, -17.28) mm, rotated rx 180 ry 0 rz 90 deg; joints [74.269, -18.238, 89.296, 0, 18.942, 74.269]
  MoveL 9696 to (-67.1, 31.4, -17.69) mm, rotated rx -180 ry 0 rz 90 deg; joints [74.218, -18.223, 89.311, 0, 18.912, 74.218]
  MoveL 9697 to (-67.6, 29.96, -18.09) mm, rotated rx 180 ry 0 rz 90 deg; joints [74.165, -18.203, 89.304, 0, 18.9, 74.165]
  MoveL 9698 to (-67.74, 28.46, -18.5) mm, rotated rx 180 ry 0 rz 90 deg; joints [74.112, -18.178, 89.27, 0, 18.908, 74.112]
  MoveL 9699 to (-67.74, 7.58, -18.5) mm, rotated rx 180 ry 0 rz 90 deg; joints [73.409, -18.087, 88.862, 0, 19.225, 73.409]
  MoveL 9700 to (-67.74, 7.11, -18.5) mm, rotated rx 180 ry 0 rz 90 deg; joints [73.393, -18.085, 88.853, 0, 19.233, 73.393]
  MoveL 9701 to (-67.68, 6.63, -18.5) mm, rotated rx 180 ry 0 rz 90 deg; joints [73.377, -18.082, 88.839, 0, 19.243, 73.377]
  MoveC 9702 to (-66.79, 5.46, -18.5) mm, rotated rx 180 ry 0 rz 90 deg; joints [73.347, -18.064, 88.756, 0, 19.308, 73.347] to (-65.39, 5.02, -18.5) mm, rotated rx -180 ry 0 rz 90 deg; joints [73.346, -18.04, 88.652, 0, 19.388, 73.346]
  MoveL 9703 to (-64.91, 5.1, -18.5) mm, rotated rx -180 ry 0 rz 90 deg; joints [73.354, -18.034, 88.622, 0, 19.411, 73.354]
  MoveL 9704 to (-61.12, 6.04, -18.5) mm, rotated rx 180 ry 0 rz 90 deg; joints [73.423, -17.98, 88.386, 0, 19.595, 73.423]
  MoveL 9705 to (-44.07, 10.43, -18.5) mm, rotated rx 180 ry 0 rz 90 deg; joints [73.737, -17.733, 87.315, 0, 20.418, 73.737]
  MoveL 9706 to (-40.34, 11.41, -18.5) mm, rotated rx 180 ry 0 rz 90 deg; joints [73.805, -17.677, 87.079, 0, 20.599, 73.805]
  MoveL 9707 to (-40.34, 34.88, -18.5) mm, rotated rx 180 ry 0 rz 90 deg; joints [74.586, -17.784, 87.534, 0, 20.25, 74.586]
  MoveC 9708 to (-52.37, 43.01, -18.5) mm, rotated rx 180 ry 0 rz 90 deg; joints [74.748, -18.008, 88.507, 0, 19.501, 74.748] to (-64.44, 51.08, -18.5) mm, rotated rx 180 ry 0 rz 90 deg; joints [74.911, -18.222, 89.47, 0, 18.752, 74.911]
  MoveC 9709 to (-66.38, 50.92, -18.5) mm, rotated rx -180 ry 0 rz 90 deg; joints [74.887, -18.249, 89.597, 0, 18.653, 74.887] to (-67.74, 49.53, -18.5) mm, rotated rx 180 ry 0 rz 90 deg; joints [74.828, -18.264, 89.663, 0, 18.601, 74.828]
  MoveL 9710 to (-67.74, 48.8, -18.5) mm, rotated rx 180 ry 0 rz 90 deg; joints [74.803, -18.261, 89.65, 0, 18.611, 74.803]
  MoveL 9711 to (-67.74, 28.46, -18.5) mm, rotated rx 180 ry 0 rz 90 deg; joints [74.112, -18.178, 89.27, 0, 18.908, 74.112]
  MoveL 9712 to (-60.19, 28.46, -18.5) mm, rotated rx -180 ry 0 rz 90 deg; joints [74.185, -18.065, 88.762, 0, 19.303, 74.185]
  MoveL 9713 to (-60.19, 28.46, -15.5) mm, rotated rx 180 ry 0 rz 90 deg; joints [74.185, -18.222, 88.866, 0, 19.356, 74.185]
  Establecer velocidad (1000.0 mm/s)
  MoveL 9714 to (-60.19, 28.46, 10) mm, rotated rx 180 ry 0 rz 90 deg; joints [74.185, -19.553, 89.724, 0, 19.829, 74.185]
  Establecer velocidad (66.7 mm/s)
  MoveL 9715 to (-48.57, -54.96, 10) mm, rotated rx -180 ry 0 rz 90 deg; joints [71.542, -18.944, 87.186, 0, 21.758, 71.542]
  MoveL 9716 to (-48.57, -54.96, -15.25) mm, rotated rx -180 ry 0 rz 90 deg; joints [71.542, -17.641, 86.336, 0, 21.304, 71.542]
  MoveL 9717 to (-47.07, -55.15, -15.66) mm, rotated rx 180 ry 0 rz 90 deg; joints [71.552, -17.594, 86.215, 0, 21.379, 71.552]
  MoveL 9718 to (-45.56, -54.96, -16.06) mm, rotated rx 180 ry 0 rz 90 deg; joints [71.574, -17.549, 86.102, 0, 21.446, 71.574]
  MoveL 9719 to (-44.13, -54.45, -16.47) mm, rotated rx -180 ry 0 rz 90 deg; joints [71.606, -17.506, 86.002, 0, 21.505, 71.606]
  MoveL 9720 to (-42.85, -53.64, -16.88) mm, rotated rx 180 ry 0 rz 90 deg; joints [71.647, -17.468, 85.918, 0, 21.55, 71.647]
  MoveL 9721 to (-41.78, -52.56, -17.28) mm, rotated rx 180 ry 0 rz 90 deg; joints [71.693, -17.435, 85.855, 0, 21.58, 71.693]
  MoveL 9722 to (-40.97, -51.27, -17.69) mm, rotated rx 180 ry 0 rz 90 deg; joints [71.744, -17.408, 85.815, 0, 21.593, 71.744]
  MoveL 9723 to (-40.47, -49.83, -18.09) mm, rotated rx 180 ry 0 rz 90 deg; joints [71.796, -17.387, 85.8, 0, 21.587, 71.796]
  MoveL 9724 to (-40.34, -48.32, -18.5) mm, rotated rx -180 ry 0 rz 90 deg; joints [71.846, -17.372, 85.81, 0, 21.562, 71.846]
  MoveL 9725 to (-40.34, -29.67, -18.5) mm, rotated rx 180 ry 0 rz 90 deg; joints [72.453, -17.473, 86.223, 0, 21.249, 72.453]
  MoveL 9726 to (-43.12, -30.18, -18.5) mm, rotated rx 180 ry 0 rz 90 deg; joints [72.408, -17.516, 86.403, 0, 21.113, 72.408]
  MoveL 9727 to (-62.07, -33.69, -18.5) mm, rotated rx 180 ry 0 rz 90 deg; joints [72.093, -17.804, 87.617, 0, 20.187, 72.093]
  MoveL 9728 to (-66, -34.45, -18.5) mm, rotated rx 180 ry 0 rz 90 deg; joints [72.026, -17.861, 87.865, 0, 19.996, 72.026]
  MoveC 9729 to (-67.23, -35.17, -18.5) mm, rotated rx 180 ry 0 rz 90 deg; joints [71.989, -17.877, 87.932, 0, 19.944, 71.989] to (-67.73, -36.5, -18.5) mm, rotated rx 180 ry 0 rz 90 deg; joints [71.94, -17.878, 87.937, 0, 19.941, 71.94]
  MoveL 9730 to (-67.74, -36.96, -18.5) mm, rotated rx 180 ry 0 rz 90 deg; joints [71.925, -17.875, 87.928, 0, 19.948, 71.925]
  MoveL 9731 to (-67.74, -65.66, -18.5) mm, rotated rx -180 ry 0 rz 90 deg; joints [70.981, -17.725, 87.279, 0, 20.446, 70.981]
  MoveC 9732 to (-67.11, -67.19, -18.5) mm, rotated rx 180 ry 0 rz 90 deg; joints [70.938, -17.706, 87.201, 0, 20.505, 70.938] to (-65.59, -67.82, -18.5) mm, rotated rx 180 ry 0 rz 90 deg; joints [70.935, -17.679, 87.084, 0, 20.595, 70.935]
  MoveC 9733 to (-65.22, -67.82, -18.5) mm, rotated rx -180 ry 0 rz 90 deg; joints [70.939, -17.673, 87.059, 0, 20.614, 70.939] to (-64.86, -67.81, -18.5) mm, rotated rx -180 ry 0 rz 90 deg; joints [70.943, -17.667, 87.035, 0, 20.632, 70.943]
  MoveC 9734 to (-52.6, -67.43, -18.5) mm, rotated rx 180 ry 0 rz 90 deg; joints [71.093, -17.47, 86.211, 0, 21.259, 71.093] to (-40.34, -66.97, -18.5) mm, rotated rx 180 ry 0 rz 90 deg; joints [71.243, -17.266, 85.382, 0, 21.885, 71.243]
  MoveL 9735 to (-40.34, -48.32, -18.5) mm, rotated rx -180 ry 0 rz 90 deg; joints [71.846, -17.372, 85.81, 0, 21.562, 71.846]
  MoveL 9736 to (-47.88, -48.32, -18.5) mm, rotated rx -180 ry 0 rz 90 deg; joints [71.765, -17.498, 86.328, 0, 21.17, 71.765]
